LIN {X 0,Y 238.565,Z 456.874,A -85,B 0,C 180,E1 -19550.701,E2 -19550.701} C_VEL
LIN {X 0,Y 241.685,Z 448.178,A -85,B 0,C 180,E1 -19554.022,E2 -19554.022} C_VEL
LIN {X 0,Y 244.667,Z 440.384,A -85,B 0,C 180,E1 -19556.437,E2 -19556.437} C_VEL
LIN {X 0,Y 247.814,Z 431.182,A -85,B 0,C 180,E1 -19558.823,E2 -19558.823} C_VEL
LIN {X 0,Y 251.41,Z 420.34,A -85,B 0,C 180,E1 -19561.14,E2 -19561.14} C_VEL
LIN {X 0,Y 255.12,Z 408.504,A -85,B 0,C 180,E1 -19563.195,E2 -19563.195} C_VEL
LIN {X 0,Y 257.974,Z 398.718,A -85,B 0,C 180,E1 -19564.607,E2 -19564.607} C_VEL
LIN {X 0,Y 257.894,Z 393.482,A -85,B 0,C 180,E1 -19565.491,E2 -19565.491} C_VEL
LIN {X 0,Y 256.687,Z 381.828,A -85,B 0,C 180,E1 -19567.439,E2 -19567.439} C_VEL
LIN {X 0,Y 254.25,Z 368.563,A -85,B 0,C 180,E1 -19569.568,E2 -19569.568} C_VEL
LIN {X 0,Y 250.278,Z 354.47,A -85,B 0,C 180,E1 -19571.817,E2 -19571.817} C_VEL
LIN {X 0,Y 245.396,Z 341.798,A -85,B 0,C 180,E1 -19573.907,E2 -19573.907} C_VEL
LIN {X 0,Y 241.213,Z 333.323,A -85,B 0,C 180,E1 -19575.435,E2 -19575.435} C_VEL
LIN {X 0,Y 239.306,Z 329.7,A -85,B 0,C 180,E1 -19576.09,E2 -19576.09} C_VEL
LIN {X 0,Y 236.728,Z 325.904,A -85,B 0,C 180,E1 -19576.935,E2 -19576.935} C_VEL
LIN {X 0,Y 236.107,Z 323.82,A -85,B 0,C 180,E1 -19577.26,E2 -19577.26} C_VEL
LIN {X 0,Y 235.752,Z 321.234,A -85,B 0,C 180,E1 -19581.242,E2 -19581.242} C_VEL
LIN {X 0,Y 235.353,Z 318.757,A -85,B 0,C 180,E1 -19585.433,E2 -19585.433} C_VEL
LIN {X 0,Y 235.026,Z 316.609,A -85,B 0,C 180,E1 -19589.446,E2 -19589.446} C_VEL
LIN {X 0,Y 234.932,Z 315.851,A -85,B 0,C 180,E1 -19591.404,E2 -19591.404} C_VEL
LIN {X 0,Y 234.982,Z 315.842,A -85,B 0,C 180,E1 -19595.246,E2 -19595.246} C_VEL
LIN {X 0,Y 235.006,Z 315.837,A -85,B 0,C 180,E1 -19598.97,E2 -19598.97} C_VEL
LIN {X 0,Y 235.091,Z 315.823,A -85,B 0,C 180,E1 -19603.059,E2 -19603.059} C_VEL
LIN {X 0,Y 235.103,Z 315.821,A -85,B 0,C 180,E1 -19607.922,E2 -19607.922} C_VEL
LIN {X 0,Y 235.305,Z 315.795,A -85,B 0,C 180,E1 -19611.412,E2 -19611.412} C_VEL
LIN {X 0,Y 235.2,Z 315.808,A -85,B 0,C 180,E1 -19614.857,E2 -19614.857} C_VEL
LIN {X 0,Y 235.588,Z 315.759,A -85,B 0,C 180,E1 -19618.291,E2 -19618.291} C_VEL
LIN {X 0,Y 235.588,Z 315.764,A -85,B 0,C 180,E1 -19621.71,E2 -19621.71} C_VEL
LIN {X 0,Y 235.344,Z 315.795,A -85,B 0,C 180,E1 -19626.861,E2 -19626.861} C_VEL
LIN {X 0,Y 235.208,Z 315.813,A -85,B 0,C 180,E1 -19630.328,E2 -19630.328} C_VEL
LIN {X 0,Y 235.107,Z 315.822,A -85,B 0,C 180,E1 -19635.607,E2 -19635.607} C_VEL
LIN {X 0,Y 235.004,Z 315.838,A -85,B 0,C 180,E1 -19639.206,E2 -19639.206} C_VEL
LIN {X 0,Y 234.956,Z 315.845,A -85,B 0,C 180,E1 -19642.883,E2 -19642.883} C_VEL
LIN {X 0,Y 234.963,Z 315.84,A -85,B 0,C 180,E1 -19646.658,E2 -19646.658} C_VEL
LIN {X 0,Y 234.918,Z 315.843,A -85,B 0,C 180,E1 -19650.57,E2 -19650.57} C_VEL
LIN {X 0,Y 234.939,Z 315.84,A -85,B 0,C 180,E1 -19653.115,E2 -19653.115} C_VEL
LIN {X 0,Y 235.197,Z 317.589,A -85,B 0,C 180,E1 -19656.7,E2 -19656.7} C_VEL
LIN {X 0,Y 235.53,Z 319.939,A -85,B 0,C 180,E1 -19661.031,E2 -19661.031} C_VEL
LIN {X 0,Y 235.683,Z 321.16,A -85,B 0,C 180,E1 -19662.76,E2 -19662.76} C_VEL
LIN {X 0,Y 236.839,Z 324.025,A -85,B 0,C 180,E1 -19663.204,E2 -19663.204} C_VEL
LIN {X 0,Y 238.973,Z 326.929,A -85,B 0,C 180,E1 -19663.895,E2 -19663.895} C_VEL
LIN {X 0,Y 240.953,Z 330.465,A -85,B 0,C 180,E1 -19664.575,E2 -19664.575} C_VEL
LIN {X 0,Y 245.815,Z 339.929,A -85,B 0,C 180,E1 -19666.354,E2 -19666.354} C_VEL
LIN {X 0,Y 250.518,Z 351.507,A -85,B 0,C 180,E1 -19668.337,E2 -19668.337} C_VEL
LIN {X 0,Y 254.323,Z 363.793,A -85,B 0,C 180,E1 -19670.381,E2 -19670.381} C_VEL
LIN {X 0,Y 257.065,Z 376.3,A -85,B 0,C 180,E1 -19672.452,E2 -19672.452} C_VEL
LIN {X 0,Y 258.779,Z 388.609,A -85,B 0,C 180,E1 -19674.563,E2 -19674.563} C_VEL
LIN {X 0,Y 258.908,Z 392.584,A -85,B 0,C 180,E1 -19675.248,E2 -19675.248} C_VEL
LIN {X 0,Y 255.3,Z 405.294,A -85,B 0,C 180,E1 -19677.066,E2 -19677.066} C_VEL
LIN {X 0,Y 251.996,Z 415.961,A -85,B 0,C 180,E1 -19678.94,E2 -19678.94} C_VEL
LIN {X 0,Y 248.366,Z 427.006,A -85,B 0,C 180,E1 -19681.307,E2 -19681.307} C_VEL
LIN {X 0,Y 244.682,Z 437.336,A -85,B 0,C 180,E1 -19684.023,E2 -19684.023} C_VEL
LIN {X 0,Y 241.427,Z 446.098,A -85,B 0,C 180,E1 -19686.86,E2 -19686.86} C_VEL
LIN {X 0,Y 239.063,Z 452.429,A -85,B 0,C 180,E1 -19689.344,E2 -19689.344} C_VEL
LIN {X 0,Y 236.617,Z 459.393,A -85,B 0,C 180,E1 -19692.722,E2 -19692.722} C_VEL
LIN {X 0,Y 234.756,Z 464.865,A -85,B 0,C 180,E1 -19696.144,E2 -19696.144} C_VEL
LIN {X 0,Y 233.633,Z 468.994,A -85,B 0,C 180,E1 -19699.603,E2 -19699.603} C_VEL
LIN {X 0,Y 232.937,Z 471.894,A -85,B 0,C 180,E1 -19703.069,E2 -19703.069} C_VEL
LIN {X 0,Y 232.691,Z 473.635,A -85,B 0,C 180,E1 -19706.538,E2 -19706.538} C_VEL
LIN {X 0,Y 232.72,Z 474.241,A -85,B 0,C 180,E1 -19710.001,E2 -19710.001} C_VEL
LIN {X 0,Y 232.691,Z 473.672,A -85,B 0,C 180,E1 -19713.464,E2 -19713.464} C_VEL
LIN {X 0,Y 232.921,Z 471.98,A -85,B 0,C 180,E1 -19716.933,E2 -19716.933} C_VEL
LIN {X 0,Y 233.606,Z 469.125,A -85,B 0,C 180,E1 -19720.4,E2 -19720.4} C_VEL
LIN {X 0,Y 234.736,Z 465.04,A -85,B 0,C 180,E1 -19723.859,E2 -19723.859} C_VEL
LIN {X 0,Y 236.558,Z 459.624,A -85,B 0,C 180,E1 -19727.284,E2 -19727.284} C_VEL
LIN {X 0,Y 239.001,Z 452.724,A -85,B 0,C 180,E1 -19730.663,E2 -19730.663} C_VEL
LIN {X 0,Y 242.204,Z 444.112,A -85,B 0,C 180,E1 -19733.969,E2 -19733.969} C_VEL
LIN {X 0,Y 245.639,Z 434.956,A -85,B 0,C 180,E1 -19736.784,E2 -19736.784} C_VEL
LIN {X 0,Y 248.854,Z 425.634,A -85,B 0,C 180,E1 -19739.155,E2 -19739.155} C_VEL
LIN {X 0,Y 252.888,Z 413.567,A -85,B 0,C 180,E1 -19741.638,E2 -19741.638} C_VEL
LIN {X 0,Y 256.604,Z 401.244,A -85,B 0,C 180,E1 -19743.684,E2 -19743.684} C_VEL
LIN {X 0,Y 259.081,Z 391.806,A -85,B 0,C 180,E1 -19744.989,E2 -19744.989} C_VEL
LIN {X 0,Y 257.665,Z 379.68,A -85,B 0,C 180,E1 -19747.112,E2 -19747.112} C_VEL
LIN {X 0,Y 255.437,Z 368.067,A -85,B 0,C 180,E1 -19749.052,E2 -19749.052} C_VEL
LIN {X 0,Y 251.911,Z 355.507,A -85,B 0,C 180,E1 -19751.126,E2 -19751.126} C_VEL
LIN {X 0,Y 247.397,Z 343.495,A -85,B 0,C 180,E1 -19753.173,E2 -19753.173} C_VEL
LIN {X 0,Y 244.519,Z 337.246,A -85,B 0,C 180,E1 -19754.3,E2 -19754.3} C_VEL
LIN {X 0,Y 240.718,Z 330.109,A -85,B 0,C 180,E1 -19755.662,E2 -19755.662} C_VEL
LIN {X 0,Y 238.456,Z 326.031,A -85,B 0,C 180,E1 -19756.441,E2 -19756.441} C_VEL
LIN {X 0,Y 236.365,Z 323.227,A -85,B 0,C 180,E1 -19757.123,E2 -19757.123} C_VEL
LIN {X 0,Y 235.632,Z 320.937,A -85,B 0,C 180,E1 -19757.444,E2 -19757.444} C_VEL
LIN {X 0,Y 235.376,Z 318.821,A -85,B 0,C 180,E1 -19761.168,E2 -19761.168} C_VEL
LIN {X 0,Y 235.047,Z 316.644,A -85,B 0,C 180,E1 -19765.381,E2 -19765.381} C_VEL
LIN {X 0,Y 234.953,Z 315.845,A -85,B 0,C 180,E1 -19767.423,E2 -19767.423} C_VEL
LIN {X 0,Y 234.902,Z 315.849,A -85,B 0,C 180,E1 -19771.399,E2 -19771.399} C_VEL
LIN {X 0,Y 234.953,Z 315.841,A -85,B 0,C 180,E1 -19775.243,E2 -19775.243} C_VEL
LIN {X 0,Y 234.997,Z 315.838,A -85,B 0,C 180,E1 -19778.968,E2 -19778.968} C_VEL
LIN {X 0,Y 235.097,Z 315.822,A -85,B 0,C 180,E1 -19783.059,E2 -19783.059} C_VEL
LIN {X 0,Y 235.103,Z 315.821,A -85,B 0,C 180,E1 -19787.921,E2 -19787.921} C_VEL
LIN {X 0,Y 235.311,Z 315.798,A -85,B 0,C 180,E1 -19791.411,E2 -19791.411} C_VEL
LIN {X 0,Y 235.205,Z 315.813,A -85,B 0,C 180,E1 -19794.857,E2 -19794.857} C_VEL
LIN {X 0,Y 235.593,Z 315.765,A -85,B 0,C 180,E1 -19798.29,E2 -19798.29} C_VEL
LIN {X 0,Y 235.593,Z 315.764,A -85,B 0,C 180,E1 -19801.709,E2 -19801.709} C_VEL
LIN {X 0,Y 235.354,Z 315.792,A -85,B 0,C 180,E1 -19806.86,E2 -19806.86} C_VEL
LIN {X 0,Y 235.214,Z 315.812,A -85,B 0,C 180,E1 -19810.327,E2 -19810.327} C_VEL
LIN {X 0,Y 235.113,Z 315.824,A -85,B 0,C 180,E1 -19815.606,E2 -19815.606} C_VEL
LIN {X 0,Y 235.007,Z 315.837,A -85,B 0,C 180,E1 -19819.206,E2 -19819.206} C_VEL
LIN {X 0,Y 234.952,Z 315.844,A -85,B 0,C 180,E1 -19822.884,E2 -19822.884} C_VEL
LIN {X 0,Y 234.967,Z 315.843,A -85,B 0,C 180,E1 -19826.657,E2 -19826.657} C_VEL
LIN {X 0,Y 234.936,Z 315.851,A -85,B 0,C 180,E1 -19828.596,E2 -19828.596} C_VEL
LIN {X 0,Y 235.236,Z 317.68,A -85,B 0,C 180,E1 -19832.532,E2 -19832.532} C_VEL
LIN {X 0,Y 235.552,Z 319.993,A -85,B 0,C 180,E1 -19836.636,E2 -19836.636} C_VEL
LIN {X 0,Y 235.948,Z 322.582,A -85,B 0,C 180,E1 -19840.793,E2 -19840.793} C_VEL
LIN {X 0,Y 236.179,Z 323.866,A -85,B 0,C 180,E1 -19841.659,E2 -19841.659} C_VEL
LIN {X 0,Y 236.561,Z 326.147,A -85,B 0,C 180,E1 -19842.401,E2 -19842.401} C_VEL
LIN {X 0,Y 237.321,Z 330.696,A -85,B 0,C 180,E1 -19843.304,E2 -19843.304} C_VEL
LIN {X 0,Y 240.561,Z 345.361,A -85,B 0,C 180,E1 -19845.198,E2 -19845.198} C_VEL
LIN {X 0,Y 241.142,Z 347.057,A -85,B 0,C 180,E1 -19845.474,E2 -19845.474} C_VEL
LIN {X 0,Y 244.976,Z 357.702,A -85,B 0,C 180,E1 -19847.338,E2 -19847.338} C_VEL
LIN {X 0,Y 248.398,Z 370.303,A -85,B 0,C 180,E1 -19849.467,E2 -19849.467} C_VEL
LIN {X 0,Y 250.733,Z 383.447,A -85,B 0,C 180,E1 -19851.705,E2 -19851.705} C_VEL
LIN {X 0,Y 251.803,Z 394.831,A -85,B 0,C 180,E1 -19853.714,E2 -19853.714} C_VEL
LIN {X 0,Y 251.861,Z 399.873,A -85,B 0,C 180,E1 -19854.61,E2 -19854.61} C_VEL
LIN {X 0,Y 248.134,Z 412.127,A -85,B 0,C 180,E1 -19856.475,E2 -19856.475} C_VEL
LIN {X 0,Y 244.065,Z 424.3,A -85,B 0,C 180,E1 -19858.78,E2 -19858.78} C_VEL
LIN {X 0,Y 240.312,Z 434.52,A -85,B 0,C 180,E1 -19861.149,E2 -19861.149} C_VEL
LIN {X 0,Y 236.728,Z 444.502,A -85,B 0,C 180,E1 -19864.03,E2 -19864.03} C_VEL
LIN {X 0,Y 233.466,Z 452.792,A -85,B 0,C 180,E1 -19866.962,E2 -19866.962} C_VEL
LIN {X 0,Y 230.488,Z 460.579,A -85,B 0,C 180,E1 -19870.402,E2 -19870.402} C_VEL
LIN {X 0,Y 228.359,Z 466.775,A -85,B 0,C 180,E1 -19873.919,E2 -19873.919} C_VEL
LIN {X 0,Y 226.816,Z 471.566,A -85,B 0,C 180,E1 -19877.473,E2 -19877.473} C_VEL
LIN {X 0,Y 225.98,Z 475.077,A -85,B 0,C 180,E1 -19881.054,E2 -19881.054} C_VEL
LIN {X 0,Y 225.589,Z 477.385,A -85,B 0,C 180,E1 -19884.637,E2 -19884.637} C_VEL
LIN {X 0,Y 225.545,Z 478.545,A -85,B 0,C 180,E1 -19888.214,E2 -19888.214} C_VEL
LIN {X 0,Y 225.631,Z 478.698,A -85,B 0,C 180,E1 -19889.999,E2 -19889.999} C_VEL
LIN {X 0,Y 225.522,Z 478.094,A -85,B 0,C 180,E1 -19893.573,E2 -19893.573} C_VEL
LIN {X 0,Y 225.734,Z 476.348,A -85,B 0,C 180,E1 -19897.153,E2 -19897.153} C_VEL
LIN {X 0,Y 226.336,Z 473.435,A -85,B 0,C 180,E1 -19900.736,E2 -19900.736} C_VEL
LIN {X 0,Y 227.557,Z 469.287,A -85,B 0,C 180,E1 -19904.304,E2 -19904.304} C_VEL
LIN {X 0,Y 229.363,Z 463.793,A -85,B 0,C 180,E1 -19907.842,E2 -19907.842} C_VEL
LIN {X 0,Y 231.889,Z 456.803,A -85,B 0,C 180,E1 -19911.326,E2 -19911.326} C_VEL
LIN {X 0,Y 235.171,Z 448.107,A -85,B 0,C 180,E1 -19914.732,E2 -19914.732} C_VEL
LIN {X 0,Y 238.269,Z 440.313,A -85,B 0,C 180,E1 -19917.205,E2 -19917.205} C_VEL
LIN {X 0,Y 242.163,Z 429.475,A -85,B 0,C 180,E1 -19920.04,E2 -19920.04} C_VEL
LIN {X 0,Y 246.341,Z 417.287,A -85,B 0,C 180,E1 -19922.58,E2 -19922.58} C_VEL
LIN {X 0,Y 250.239,Z 405.245,A -85,B 0,C 180,E1 -19924.586,E2 -19924.586} C_VEL
LIN {X 0,Y 251.755,Z 399.909,A -85,B 0,C 180,E1 -19925.354,E2 -19925.354} C_VEL
LIN {X 0,Y 251.35,Z 389.821,A -85,B 0,C 180,E1 -19927.147,E2 -19927.147} C_VEL
LIN {X 0,Y 249.87,Z 378.381,A -85,B 0,C 180,E1 -19929.135,E2 -19929.135} C_VEL
LIN {X 0,Y 247.702,Z 367.848,A -85,B 0,C 180,E1 -19930.905,E2 -19930.905} C_VEL
LIN {X 0,Y 244.696,Z 356.943,A -85,B 0,C 180,E1 -19932.745,E2 -19932.745} C_VEL
LIN {X 0,Y 240.512,Z 345.764,A -85,B 0,C 180,E1 -19934.713,E2 -19934.713} C_VEL
LIN {X 0,Y 236.668,Z 337.699,A -85,B 0,C 180,E1 -19936.263,E2 -19936.263} C_VEL
LIN {X 0,Y 234.508,Z 333.706,A -85,B 0,C 180,E1 -19937.089,E2 -19937.089} C_VEL
LIN {X 0,Y 232.407,Z 330.075,A -85,B 0,C 180,E1 -19937.86,E2 -19937.86} C_VEL
LIN {X 0,Y 231.653,Z 328.876,A -85,B 0,C 180,E1 -19938.13,E2 -19938.13} C_VEL
LIN {X 0,Y 229.64,Z 325.946,A -85,B 0,C 180,E1 -19938.853,E2 -19938.853} C_VEL
LIN {X 0,Y 228.973,Z 323.734,A -85,B 0,C 180,E1 -19939.217,E2 -19939.217} C_VEL
LIN {X 0,Y 228.476,Z 320.749,A -85,B 0,C 180,E1 -19944.236,E2 -19944.236} C_VEL
LIN {X 0,Y 228.14,Z 318.506,A -85,B 0,C 180,E1 -19948.42,E2 -19948.42} C_VEL
LIN {X 0,Y 227.874,Z 316.729,A -85,B 0,C 180,E1 -19952.444,E2 -19952.444} C_VEL
LIN {X 0,Y 227.909,Z 316.72,A -85,B 0,C 180,E1 -19956.367,E2 -19956.367} C_VEL
LIN {X 0,Y 227.937,Z 316.715,A -85,B 0,C 180,E1 -19960.174,E2 -19960.174} C_VEL
LIN {X 0,Y 228.051,Z 316.704,A -85,B 0,C 180,E1 -19963.898,E2 -19963.898} C_VEL
LIN {X 0,Y 228.062,Z 316.699,A -85,B 0,C 180,E1 -19967.543,E2 -19967.543} C_VEL
LIN {X 0,Y 228.246,Z 316.674,A -85,B 0,C 180,E1 -19971.144,E2 -19971.144} C_VEL
LIN {X 0,Y 228.296,Z 316.673,A -85,B 0,C 180,E1 -19972.927,E2 -19972.927} C_VEL
LIN {X 0,Y 228.547,Z 316.636,A -85,B 0,C 180,E1 -19978.238,E2 -19978.238} C_VEL
LIN {X 0,Y 228.547,Z 316.641,A -85,B 0,C 180,E1 -19981.762,E2 -19981.762} C_VEL
LIN {X 0,Y 228.296,Z 316.673,A -85,B 0,C 180,E1 -19987.073,E2 -19987.073} C_VEL
LIN {X 0,Y 228.139,Z 316.69,A -85,B 0,C 180,E1 -19990.652,E2 -19990.652} C_VEL
LIN {X 0,Y 228.055,Z 316.699,A -85,B 0,C 180,E1 -19994.273,E2 -19994.273} C_VEL
LIN {X 0,Y 227.998,Z 316.706,A -85,B 0,C 180,E1 -19997.954,E2 -19997.954} C_VEL
LIN {X 0,Y 227.925,Z 316.719,A -85,B 0,C 180,E1 -20002.33,E2 -20002.33} C_VEL
LIN {X 0,Y 227.937,Z 316.715,A -85,B 0,C 180,E1 -20006.603,E2 -20006.603} C_VEL
LIN {X 0,Y 227.893,Z 316.717,A -85,B 0,C 180,E1 -20010.292,E2 -20010.292} C_VEL
LIN {X 0,Y 227.862,Z 316.722,A -85,B 0,C 180,E1 -20011.624,E2 -20011.624} C_VEL
LIN {X 0,Y 228.139,Z 318.464,A -85,B 0,C 180,E1 -20015.825,E2 -20015.825} C_VEL
LIN {X 0,Y 228.495,Z 320.901,A -85,B 0,C 180,E1 -20020.524,E2 -20020.524} C_VEL
LIN {X 0,Y 228.578,Z 321.271,A -85,B 0,C 180,E1 -20020.796,E2 -20020.796} C_VEL
LIN {X 0,Y 229.838,Z 324.342,A -85,B 0,C 180,E1 -20021.323,E2 -20021.323} C_VEL
LIN {X 0,Y 231.924,Z 327.058,A -85,B 0,C 180,E1 -20022.054,E2 -20022.054} C_VEL
LIN {X 0,Y 234.094,Z 330.783,A -85,B 0,C 180,E1 -20022.859,E2 -20022.859} C_VEL
LIN {X 0,Y 235.185,Z 332.597,A -85,B 0,C 180,E1 -20023.27,E2 -20023.27} C_VEL
LIN {X 0,Y 239.558,Z 340.943,A -85,B 0,C 180,E1 -20024.983,E2 -20024.983} C_VEL
LIN {X 0,Y 243.811,Z 350.913,A -85,B 0,C 180,E1 -20026.854,E2 -20026.854} C_VEL
LIN {X 0,Y 247.435,Z 362.038,A -85,B 0,C 180,E1 -20028.826,E2 -20028.826} C_VEL
LIN {X 0,Y 250.277,Z 373.956,A -85,B 0,C 180,E1 -20030.896,E2 -20030.896} C_VEL
LIN {X 0,Y 252.067,Z 385.053,A -85,B 0,C 180,E1 -20032.884,E2 -20032.884} C_VEL
LIN {X 0,Y 252.732,Z 394.02,A -85,B 0,C 180,E1 -20034.505,E2 -20034.505} C_VEL
LIN {X 0,Y 248.996,Z 406.539,A -85,B 0,C 180,E1 -20036.365,E2 -20036.365} C_VEL
LIN {X 0,Y 245.266,Z 417.98,A -85,B 0,C 180,E1 -20038.471,E2 -20038.471} C_VEL
LIN {X 0,Y 241.896,Z 427.696,A -85,B 0,C 180,E1 -20040.647,E2 -20040.647} C_VEL
LIN {X 0,Y 238.299,Z 437.407,A -85,B 0,C 180,E1 -20043.273,E2 -20043.273} C_VEL
LIN {X 0,Y 234.867,Z 446.17,A -85,B 0,C 180,E1 -20046.175,E2 -20046.175} C_VEL
LIN {X 0,Y 232.386,Z 452.5,A -85,B 0,C 180,E1 -20048.722,E2 -20048.722} C_VEL
LIN {X 0,Y 229.807,Z 459.464,A -85,B 0,C 180,E1 -20052.193,E2 -20052.193} C_VEL
LIN {X 0,Y 227.837,Z 464.935,A -85,B 0,C 180,E1 -20055.714,E2 -20055.714} C_VEL
LIN {X 0,Y 226.612,Z 469.064,A -85,B 0,C 180,E1 -20059.277,E2 -20059.277} C_VEL
LIN {X 0,Y 225.885,Z 471.963,A -85,B 0,C 180,E1 -20062.852,E2 -20062.852} C_VEL
LIN {X 0,Y 225.606,Z 473.704,A -85,B 0,C 180,E1 -20066.429,E2 -20066.429} C_VEL
LIN {X 0,Y 225.636,Z 474.31,A -85,B 0,C 180,E1 -20070.001,E2 -20070.001} C_VEL
LIN {X 0,Y 225.605,Z 473.741,A -85,B 0,C 180,E1 -20073.573,E2 -20073.573} C_VEL
LIN {X 0,Y 225.845,Z 472.049,A -85,B 0,C 180,E1 -20077.151,E2 -20077.151} C_VEL
LIN {X 0,Y 226.586,Z 469.194,A -85,B 0,C 180,E1 -20080.726,E2 -20080.726} C_VEL
LIN {X 0,Y 227.816,Z 465.108,A -85,B 0,C 180,E1 -20084.288,E2 -20084.288} C_VEL
LIN {X 0,Y 229.751,Z 459.692,A -85,B 0,C 180,E1 -20087.812,E2 -20087.812} C_VEL
LIN {X 0,Y 232.335,Z 452.792,A -85,B 0,C 180,E1 -20091.284,E2 -20091.284} C_VEL
LIN {X 0,Y 235.672,Z 444.18,A -85,B 0,C 180,E1 -20094.677,E2 -20094.677} C_VEL
LIN {X 0,Y 239.29,Z 435.023,A -85,B 0,C 180,E1 -20097.554,E2 -20097.554} C_VEL
LIN {X 0,Y 242.649,Z 425.701,A -85,B 0,C 180,E1 -20099.975,E2 -20099.975} C_VEL
LIN {X 0,Y 246.85,Z 413.633,A -85,B 0,C 180,E1 -20102.506,E2 -20102.506} C_VEL
LIN {X 0,Y 250.725,Z 401.309,A -85,B 0,C 180,E1 -20104.585,E2 -20104.585} C_VEL
LIN {X 0,Y 252.885,Z 393.447,A -85,B 0,C 180,E1 -20105.705,E2 -20105.705} C_VEL
LIN {X 0,Y 251.603,Z 381.432,A -85,B 0,C 180,E1 -20107.917,E2 -20107.917} C_VEL
LIN {X 0,Y 249.779,Z 371.284,A -85,B 0,C 180,E1 -20109.695,E2 -20109.695} C_VEL
LIN {X 0,Y 246.555,Z 358.913,A -85,B 0,C 180,E1 -20111.867,E2 -20111.867} C_VEL
LIN {X 0,Y 242.119,Z 346.554,A -85,B 0,C 180,E1 -20114.09,E2 -20114.09} C_VEL
LIN {X 0,Y 238.454,Z 338.74,A -85,B 0,C 180,E1 -20115.623,E2 -20115.623} C_VEL
LIN {X 0,Y 236.232,Z 334.554,A -85,B 0,C 180,E1 -20116.487,E2 -20116.487} C_VEL
LIN {X 0,Y 234.378,Z 331.128,A -85,B 0,C 180,E1 -20117.206,E2 -20117.206} C_VEL
LIN {X 0,Y 232.191,Z 327.696,A -85,B 0,C 180,E1 -20118.005,E2 -20118.005} C_VEL
LIN {X 0,Y 231.476,Z 326.274,A -85,B 0,C 180,E1 -20118.28,E2 -20118.28} C_VEL
LIN {X 0,Y 229.392,Z 323.598,A -85,B 0,C 180,E1 -20119.017,E2 -20119.017} C_VEL
LIN {X 0,Y 228.507,Z 321.026,A -85,B 0,C 180,E1 -20119.443,E2 -20119.443} C_VEL
LIN {X 0,Y 228.159,Z 318.562,A -85,B 0,C 180,E1 -20124.179,E2 -20124.179} C_VEL
LIN {X 0,Y 227.856,Z 316.73,A -85,B 0,C 180,E1 -20128.375,E2 -20128.375} C_VEL
LIN {X 0,Y 227.855,Z 316.728,A -85,B 0,C 180,E1 -20132.441,E2 -20132.441} C_VEL
LIN {X 0,Y 227.895,Z 316.723,A -85,B 0,C 180,E1 -20136.365,E2 -20136.365} C_VEL
LIN {X 0,Y 227.937,Z 316.714,A -85,B 0,C 180,E1 -20140.174,E2 -20140.174} C_VEL
LIN {X 0,Y 228.058,Z 316.697,A -85,B 0,C 180,E1 -20143.898,E2 -20143.898} C_VEL
LIN {X 0,Y 228.063,Z 316.695,A -85,B 0,C 180,E1 -20147.542,E2 -20147.542} C_VEL
LIN {X 0,Y 228.252,Z 316.678,A -85,B 0,C 180,E1 -20151.144,E2 -20151.144} C_VEL
LIN {X 0,Y 228.302,Z 316.672,A -85,B 0,C 180,E1 -20152.927,E2 -20152.927} C_VEL
LIN {X 0,Y 228.552,Z 316.641,A -85,B 0,C 180,E1 -20158.238,E2 -20158.238} C_VEL
LIN {X 0,Y 228.552,Z 316.641,A -85,B 0,C 180,E1 -20161.762,E2 -20161.762} C_VEL
LIN {X 0,Y 228.307,Z 316.67,A -85,B 0,C 180,E1 -20167.073,E2 -20167.073} C_VEL
LIN {X 0,Y 228.145,Z 316.692,A -85,B 0,C 180,E1 -20170.651,E2 -20170.651} C_VEL
LIN {X 0,Y 228.064,Z 316.702,A -85,B 0,C 180,E1 -20174.272,E2 -20174.272} C_VEL
LIN {X 0,Y 228.002,Z 316.71,A -85,B 0,C 180,E1 -20177.953,E2 -20177.953} C_VEL
LIN {X 0,Y 227.916,Z 316.72,A -85,B 0,C 180,E1 -20182.321,E2 -20182.321} C_VEL
LIN {X 0,Y 227.941,Z 316.718,A -85,B 0,C 180,E1 -20186.602,E2 -20186.602} C_VEL
LIN {X 0,Y 227.878,Z 316.728,A -85,B 0,C 180,E1 -20187.556,E2 -20187.556} C_VEL
LIN {X 0,Y 228.153,Z 318.556,A -85,B 0,C 180,E1 -20191.578,E2 -20191.578} C_VEL
LIN {X 0,Y 228.484,Z 320.799,A -85,B 0,C 180,E1 -20195.762,E2 -20195.762} C_VEL
LIN {X 0,Y 228.993,Z 323.937,A -85,B 0,C 180,E1 -20200.779,E2 -20200.779} C_VEL
LIN {X 0,Y 230.128,Z 326.9,A -85,B 0,C 180,E1 -20201.259,E2 -20201.259} C_VEL
LIN {X 0,Y 232.296,Z 329.791,A -85,B 0,C 180,E1 -20202.019,E2 -20202.019} C_VEL
LIN {X 0,Y 234.381,Z 333.546,A -85,B 0,C 180,E1 -20202.793,E2 -20202.793} C_VEL
LIN {X 0,Y 235.827,Z 336.082,A -85,B 0,C 180,E1 -20203.343,E2 -20203.343} C_VEL
LIN {X 0,Y 239.693,Z 343.792,A -85,B 0,C 180,E1 -20204.869,E2 -20204.869} C_VEL
LIN {X 0,Y 241.142,Z 347.057,A -85,B 0,C 180,E1 -20205.474,E2 -20205.474} C_VEL
LIN {X 0,Y 242.393,Z 351.967,A -85,B 0,C 180,E1 -20206.193,E2 -20206.193} C_VEL
LIN {X 0,Y 242.772,Z 360.897,A -85,B 0,C 180,E1 -20207.207,E2 -20207.207} C_VEL
LIN {X 0,Y 242.613,Z 368.127,A -85,B 0,C 180,E1 -20208.029,E2 -20208.029} C_VEL
LIN {X 0,Y 243.089,Z 374.88,A -85,B 0,C 180,E1 -20209.021,E2 -20209.021} C_VEL
LIN {X 0,Y 244.917,Z 386.896,A -85,B 0,C 180,E1 -20211.179,E2 -20211.179} C_VEL
LIN {X 0,Y 245.705,Z 397.844,A -85,B 0,C 180,E1 -20213.215,E2 -20213.215} C_VEL
LIN {X 0,Y 245.682,Z 401.141,A -85,B 0,C 180,E1 -20213.842,E2 -20213.842} C_VEL
LIN {X 0,Y 241.853,Z 413.132,A -85,B 0,C 180,E1 -20215.735,E2 -20215.735} C_VEL
LIN {X 0,Y 237.987,Z 424.233,A -85,B 0,C 180,E1 -20217.889,E2 -20217.889} C_VEL
LIN {X 0,Y 234.084,Z 434.453,A -85,B 0,C 180,E1 -20220.306,E2 -20220.306} C_VEL
LIN {X 0,Y 230.314,Z 444.434,A -85,B 0,C 180,E1 -20223.25,E2 -20223.25} C_VEL
LIN {X 0,Y 226.909,Z 452.724,A -85,B 0,C 180,E1 -20226.256,E2 -20226.256} C_VEL
LIN {X 0,Y 223.745,Z 460.511,A -85,B 0,C 180,E1 -20229.786,E2 -20229.786} C_VEL
LIN {X 0,Y 221.477,Z 466.706,A -85,B 0,C 180,E1 -20233.405,E2 -20233.405} C_VEL
LIN {X 0,Y 219.84,Z 471.497,A -85,B 0,C 180,E1 -20237.068,E2 -20237.068} C_VEL
LIN {X 0,Y 218.942,Z 475.008,A -85,B 0,C 180,E1 -20240.764,E2 -20240.764} C_VEL
LIN {X 0,Y 218.5,Z 477.316,A -85,B 0,C 180,E1 -20244.462,E2 -20244.462} C_VEL
LIN {X 0,Y 218.448,Z 478.476,A -85,B 0,C 180,E1 -20248.156,E2 -20248.156} C_VEL
LIN {X 0,Y 218.53,Z 478.629,A -85,B 0,C 180,E1 -20249.999,E2 -20249.999} C_VEL
LIN {X 0,Y 218.427,Z 477.911,A -85,B 0,C 180,E1 -20254.104,E2 -20254.104} C_VEL
LIN {X 0,Y 218.653,Z 476.278,A -85,B 0,C 180,E1 -20257.386,E2 -20257.386} C_VEL
LIN {X 0,Y 219.307,Z 473.365,A -85,B 0,C 180,E1 -20261.085,E2 -20261.085} C_VEL
LIN {X 0,Y 220.619,Z 469.217,A -85,B 0,C 180,E1 -20264.764,E2 -20264.764} C_VEL
LIN {X 0,Y 222.54,Z 463.722,A -85,B 0,C 180,E1 -20268.409,E2 -20268.409} C_VEL
LIN {X 0,Y 225.223,Z 456.732,A -85,B 0,C 180,E1 -20271.99,E2 -20271.99} C_VEL
LIN {X 0,Y 228.713,Z 448.035,A -85,B 0,C 180,E1 -20275.479,E2 -20275.479} C_VEL
LIN {X 0,Y 231.906,Z 440.241,A -85,B 0,C 180,E1 -20278.016,E2 -20278.016} C_VEL
LIN {X 0,Y 235.992,Z 429.403,A -85,B 0,C 180,E1 -20280.91,E2 -20280.91} C_VEL
LIN {X 0,Y 240.359,Z 417.214,A -85,B 0,C 180,E1 -20283.496,E2 -20283.496} C_VEL
LIN {X 0,Y 244.31,Z 405.468,A -85,B 0,C 180,E1 -20285.489,E2 -20285.489} C_VEL
LIN {X 0,Y 245.578,Z 401.09,A -85,B 0,C 180,E1 -20286.137,E2 -20286.137} C_VEL
LIN {X 0,Y 245.139,Z 390.146,A -85,B 0,C 180,E1 -20288.188,E2 -20288.188} C_VEL
LIN {X 0,Y 243.619,Z 378.181,A -85,B 0,C 180,E1 -20290.359,E2 -20290.359} C_VEL
LIN {X 0,Y 241.034,Z 366.197,A -85,B 0,C 180,E1 -20292.487,E2 -20292.487} C_VEL
LIN {X 0,Y 237.382,Z 354.165,A -85,B 0,C 180,E1 -20294.676,E2 -20294.676} C_VEL
LIN {X 0,Y 233.977,Z 345.863,A -85,B 0,C 180,E1 -20296.303,E2 -20296.303} C_VEL
LIN {X 0,Y 230.381,Z 338.676,A -85,B 0,C 180,E1 -20297.846,E2 -20297.846} C_VEL
LIN {X 0,Y 227.567,Z 333.769,A -85,B 0,C 180,E1 -20298.991,E2 -20298.991} C_VEL
LIN {X 0,Y 225.577,Z 330.453,A -85,B 0,C 180,E1 -20299.785,E2 -20299.785} C_VEL
LIN {X 0,Y 224.793,Z 329.066,A -85,B 0,C 180,E1 -20300.101,E2 -20300.101} C_VEL
LIN {X 0,Y 222.568,Z 326.154,A -85,B 0,C 180,E1 -20300.962,E2 -20300.962} C_VEL
LIN {X 0,Y 221.711,Z 323.651,A -85,B 0,C 180,E1 -20301.407,E2 -20301.407} C_VEL
LIN {X 0,Y 221.383,Z 321.298,A -85,B 0,C 180,E1 -20305.626,E2 -20305.626} C_VEL
LIN {X 0,Y 221.105,Z 319.389,A -85,B 0,C 180,E1 -20309.431,E2 -20309.431} C_VEL
LIN {X 0,Y 220.889,Z 317.6,A -85,B 0,C 180,E1 -20313.549,E2 -20313.549} C_VEL
LIN {X 0,Y 220.873,Z 317.598,A -85,B 0,C 180,E1 -20317.553,E2 -20317.553} C_VEL
LIN {X 0,Y 220.979,Z 317.581,A -85,B 0,C 180,E1 -20322.571,E2 -20322.571} C_VEL
LIN {X 0,Y 221.002,Z 317.58,A -85,B 0,C 180,E1 -20327.138,E2 -20327.138} C_VEL
LIN {X 0,Y 221.188,Z 317.553,A -85,B 0,C 180,E1 -20330.859,E2 -20330.859} C_VEL
LIN {X 0,Y 221.121,Z 317.561,A -85,B 0,C 180,E1 -20334.529,E2 -20334.529} C_VEL
LIN {X 0,Y 221.505,Z 317.512,A -85,B 0,C 180,E1 -20338.182,E2 -20338.182} C_VEL
LIN {X 0,Y 221.505,Z 317.518,A -85,B 0,C 180,E1 -20341.818,E2 -20341.818} C_VEL
LIN {X 0,Y 221.234,Z 317.55,A -85,B 0,C 180,E1 -20347.3,E2 -20347.3} C_VEL
LIN {X 0,Y 221.06,Z 317.57,A -85,B 0,C 180,E1 -20350.997,E2 -20350.997} C_VEL
LIN {X 0,Y 221.011,Z 317.58,A -85,B 0,C 180,E1 -20356.63,E2 -20356.63} C_VEL
LIN {X 0,Y 220.888,Z 317.592,A -85,B 0,C 180,E1 -20360.487,E2 -20360.487} C_VEL
LIN {X 0,Y 220.863,Z 317.598,A -85,B 0,C 180,E1 -20364.436,E2 -20364.436} C_VEL
LIN {X 0,Y 220.823,Z 317.6,A -85,B 0,C 180,E1 -20368.516,E2 -20368.516} C_VEL
LIN {X 0,Y 220.835,Z 317.597,A -85,B 0,C 180,E1 -20370.768,E2 -20370.768} C_VEL
LIN {X 0,Y 221.073,Z 319.369,A -85,B 0,C 180,E1 -20374.906,E2 -20374.906} C_VEL
LIN {X 0,Y 221.382,Z 321.332,A -85,B 0,C 180,E1 -20378.584,E2 -20378.584} C_VEL
LIN {X 0,Y 222.505,Z 324.182,A -85,B 0,C 180,E1 -20379.108,E2 -20379.108} C_VEL
LIN {X 0,Y 225.015,Z 327.285,A -85,B 0,C 180,E1 -20380.071,E2 -20380.071} C_VEL
LIN {X 0,Y 226.995,Z 330.785,A -85,B 0,C 180,E1 -20380.882,E2 -20380.882} C_VEL
LIN {X 0,Y 228.278,Z 332.78,A -85,B 0,C 180,E1 -20381.4,E2 -20381.4} C_VEL
LIN {X 0,Y 231.304,Z 338.068,A -85,B 0,C 180,E1 -20382.635,E2 -20382.635} C_VEL
LIN {X 0,Y 235.398,Z 346.387,A -85,B 0,C 180,E1 -20384.437,E2 -20384.437} C_VEL
LIN {X 0,Y 239.556,Z 357.244,A -85,B 0,C 180,E1 -20386.572,E2 -20386.572} C_VEL
LIN {X 0,Y 242.91,Z 369.13,A -85,B 0,C 180,E1 -20388.785,E2 -20388.785} C_VEL
LIN {X 0,Y 245.334,Z 381.553,A -85,B 0,C 180,E1 -20391.087,E2 -20391.087} C_VEL
LIN {X 0,Y 246.592,Z 394.098,A -85,B 0,C 180,E1 -20393.481,E2 -20393.481} C_VEL
LIN {X 0,Y 246.588,Z 395.377,A -85,B 0,C 180,E1 -20393.717,E2 -20393.717} C_VEL
LIN {X 0,Y 242.751,Z 407.773,A -85,B 0,C 180,E1 -20395.63,E2 -20395.63} C_VEL
LIN {X 0,Y 238.545,Z 419.976,A -85,B 0,C 180,E1 -20397.975,E2 -20397.975} C_VEL
LIN {X 0,Y 234.831,Z 430.014,A -85,B 0,C 180,E1 -20400.357,E2 -20400.357} C_VEL
LIN {X 0,Y 230.801,Z 440.179,A -85,B 0,C 180,E1 -20403.312,E2 -20403.312} C_VEL
LIN {X 0,Y 227.429,Z 448.466,A -85,B 0,C 180,E1 -20406.315,E2 -20406.315} C_VEL
LIN {X 0,Y 224.304,Z 456.251,A -85,B 0,C 180,E1 -20409.84,E2 -20409.84} C_VEL
LIN {X 0,Y 221.948,Z 462.446,A -85,B 0,C 180,E1 -20413.443,E2 -20413.443} C_VEL
LIN {X 0,Y 220.176,Z 467.23,A -85,B 0,C 180,E1 -20417.09,E2 -20417.09} C_VEL
LIN {X 0,Y 219.129,Z 470.732,A -85,B 0,C 180,E1 -20420.773,E2 -20420.773} C_VEL
LIN {X 0,Y 218.601,Z 473.045,A -85,B 0,C 180,E1 -20424.466,E2 -20424.466} C_VEL
LIN {X 0,Y 218.489,Z 474.222,A -85,B 0,C 180,E1 -20428.157,E2 -20428.157} C_VEL
LIN {X 0,Y 218.536,Z 474.379,A -85,B 0,C 180,E1 -20430.001,E2 -20430.001} C_VEL
LIN {X 0,Y 218.504,Z 473.81,A -85,B 0,C 180,E1 -20433.689,E2 -20433.689} C_VEL
LIN {X 0,Y 218.795,Z 472.118,A -85,B 0,C 180,E1 -20437.383,E2 -20437.383} C_VEL
LIN {X 0,Y 219.584,Z 469.262,A -85,B 0,C 180,E1 -20441.072,E2 -20441.072} C_VEL
LIN {X 0,Y 220.916,Z 465.176,A -85,B 0,C 180,E1 -20444.745,E2 -20444.745} C_VEL
LIN {X 0,Y 222.954,Z 459.76,A -85,B 0,C 180,E1 -20448.375,E2 -20448.375} C_VEL
LIN {X 0,Y 225.687,Z 452.859,A -85,B 0,C 180,E1 -20451.943,E2 -20451.943} C_VEL
LIN {X 0,Y 229.186,Z 444.247,A -85,B 0,C 180,E1 -20455.424,E2 -20455.424} C_VEL
LIN {X 0,Y 232.984,Z 435.09,A -85,B 0,C 180,E1 -20458.366,E2 -20458.366} C_VEL
LIN {X 0,Y 236.491,Z 425.767,A -85,B 0,C 180,E1 -20460.84,E2 -20460.84} C_VEL
LIN {X 0,Y 240.849,Z 413.699,A -85,B 0,C 180,E1 -20463.42,E2 -20463.42} C_VEL
LIN {X 0,Y 244.839,Z 401.593,A -85,B 0,C 180,E1 -20465.495,E2 -20465.495} C_VEL
LIN {X 0,Y 246.608,Z 395.768,A -85,B 0,C 180,E1 -20466.342,E2 -20466.342} C_VEL
LIN {X 0,Y 245.919,Z 386.077,A -85,B 0,C 180,E1 -20468.196,E2 -20468.196} C_VEL
LIN {X 0,Y 244.255,Z 375.04,A -85,B 0,C 180,E1 -20470.263,E2 -20470.263} C_VEL
LIN {X 0,Y 241.179,Z 362.238,A -85,B 0,C 180,E1 -20472.625,E2 -20472.625} C_VEL
LIN {X 0,Y 236.697,Z 349.286,A -85,B 0,C 180,E1 -20475.111,E2 -20475.111} C_VEL
LIN {X 0,Y 232.649,Z 340.483,A -85,B 0,C 180,E1 -20476.958,E2 -20476.958} C_VEL
LIN {X 0,Y 229.811,Z 335.48,A -85,B 0,C 180,E1 -20478.139,E2 -20478.139} C_VEL
LIN {X 0,Y 227.348,Z 331.208,A -85,B 0,C 180,E1 -20479.156,E2 -20479.156} C_VEL
LIN {X 0,Y 225.189,Z 327.723,A -85,B 0,C 180,E1 -20480.027,E2 -20480.027} C_VEL
LIN {X 0,Y 224.496,Z 326.515,A -85,B 0,C 180,E1 -20480.309,E2 -20480.309} C_VEL
LIN {X 0,Y 222.352,Z 323.96,A -85,B 0,C 180,E1 -20481.134,E2 -20481.134} C_VEL
LIN {X 0,Y 221.358,Z 321.109,A -85,B 0,C 180,E1 -20481.682,E2 -20481.682} C_VEL
LIN {X 0,Y 221.073,Z 319.163,A -85,B 0,C 180,E1 -20485.746,E2 -20485.746} C_VEL
LIN {X 0,Y 220.835,Z 317.602,A -85,B 0,C 180,E1 -20489.389,E2 -20489.389} C_VEL
LIN {X 0,Y 220.876,Z 317.595,A -85,B 0,C 180,E1 -20493.547,E2 -20493.547} C_VEL
LIN {X 0,Y 220.868,Z 317.594,A -85,B 0,C 180,E1 -20497.552,E2 -20497.552} C_VEL
LIN {X 0,Y 220.985,Z 317.584,A -85,B 0,C 180,E1 -20502.571,E2 -20502.571} C_VEL
LIN {X 0,Y 221.003,Z 317.574,A -85,B 0,C 180,E1 -20507.138,E2 -20507.138} C_VEL
LIN {X 0,Y 221.194,Z 317.559,A -85,B 0,C 180,E1 -20510.859,E2 -20510.859} C_VEL
LIN {X 0,Y 221.125,Z 317.567,A -85,B 0,C 180,E1 -20514.528,E2 -20514.528} C_VEL
LIN {X 0,Y 221.51,Z 317.518,A -85,B 0,C 180,E1 -20518.182,E2 -20518.182} C_VEL
LIN {X 0,Y 221.509,Z 317.518,A -85,B 0,C 180,E1 -20521.818,E2 -20521.818} C_VEL
LIN {X 0,Y 221.244,Z 317.55,A -85,B 0,C 180,E1 -20527.3,E2 -20527.3} C_VEL
LIN {X 0,Y 221.067,Z 317.574,A -85,B 0,C 180,E1 -20530.996,E2 -20530.996} C_VEL
LIN {X 0,Y 220.995,Z 317.583,A -85,B 0,C 180,E1 -20534.739,E2 -20534.739} C_VEL
LIN {X 0,Y 220.92,Z 317.593,A -85,B 0,C 180,E1 -20538.549,E2 -20538.549} C_VEL
LIN {X 0,Y 220.884,Z 317.596,A -85,B 0,C 180,E1 -20542.675,E2 -20542.675} C_VEL
LIN {X 0,Y 220.893,Z 317.596,A -85,B 0,C 180,E1 -20546.45,E2 -20546.45} C_VEL
LIN {X 0,Y 221.141,Z 319.599,A -85,B 0,C 180,E1 -20550.899,E2 -20550.899} C_VEL
LIN {X 0,Y 221.419,Z 321.602,A -85,B 0,C 180,E1 -20554.843,E2 -20554.843} C_VEL
LIN {X 0,Y 221.706,Z 323.667,A -85,B 0,C 180,E1 -20558.532,E2 -20558.532} C_VEL
LIN {X 0,Y 222.903,Z 326.801,A -85,B 0,C 180,E1 -20559.093,E2 -20559.093} C_VEL
LIN {X 0,Y 225.343,Z 329.818,A -85,B 0,C 180,E1 -20560.023,E2 -20560.023} C_VEL
LIN {X 0,Y 227.223,Z 333.355,A -85,B 0,C 180,E1 -20560.798,E2 -20560.798} C_VEL
LIN {X 0,Y 228.538,Z 335.247,A -85,B 0,C 180,E1 -20561.315,E2 -20561.315} C_VEL
LIN {X 0,Y 230.756,Z 339.184,A -85,B 0,C 180,E1 -20562.217,E2 -20562.217} C_VEL
LIN {X 0,Y 235.178,Z 348.414,A -85,B 0,C 180,E1 -20564.151,E2 -20564.151} C_VEL
LIN {X 0,Y 238.937,Z 358.669,A -85,B 0,C 180,E1 -20566.105,E2 -20566.105} C_VEL
LIN {X 0,Y 242.295,Z 371.013,A -85,B 0,C 180,E1 -20568.323,E2 -20568.323} C_VEL
LIN {X 0,Y 243.089,Z 374.88,A -85,B 0,C 180,E1 -20569.021,E2 -20569.021} C_VEL
LIN {X 0,Y 243.414,Z 379.816,A -85,B 0,C 180,E1 -20569.789,E2 -20569.789} C_VEL
LIN {X 0,Y 242.036,Z 388.477,A -85,B 0,C 180,E1 -20570.902,E2 -20570.902} C_VEL
LIN {X 0,Y 239.847,Z 398.669,A -85,B 0,C 180,E1 -20572.329,E2 -20572.329} C_VEL
LIN {X 0,Y 239.564,Z 401.756,A -85,B 0,C 180,E1 -20572.904,E2 -20572.904} C_VEL
LIN {X 0,Y 237.965,Z 407.335,A -85,B 0,C 180,E1 -20573.795,E2 -20573.795} C_VEL
LIN {X 0,Y 234.096,Z 418.357,A -85,B 0,C 180,E1 -20575.743,E2 -20575.743} C_VEL
LIN {X 0,Y 229.887,Z 429.495,A -85,B 0,C 180,E1 -20578.173,E2 -20578.173} C_VEL
LIN {X 0,Y 226.121,Z 438.705,A -85,B 0,C 180,E1 -20580.635,E2 -20580.635} C_VEL
LIN {X 0,Y 222.865,Z 446.853,A -85,B 0,C 180,E1 -20583.296,E2 -20583.296} C_VEL
LIN {X 0,Y 219.457,Z 454.743,A -85,B 0,C 180,E1 -20586.402,E2 -20586.402} C_VEL
LIN {X 0,Y 216.348,Z 462.111,A -85,B 0,C 180,E1 -20590.057,E2 -20590.057} C_VEL
LIN {X 0,Y 214.163,Z 467.954,A -85,B 0,C 180,E1 -20593.803,E2 -20593.803} C_VEL
LIN {X 0,Y 212.875,Z 471.429,A -85,B 0,C 180,E1 -20596.637,E2 -20596.637} C_VEL
LIN {X 0,Y 211.886,Z 474.939,A -85,B 0,C 180,E1 -20600.453,E2 -20600.453} C_VEL
LIN {X 0,Y 211.405,Z 477.247,A -85,B 0,C 180,E1 -20604.276,E2 -20604.276} C_VEL
LIN {X 0,Y 211.353,Z 478.407,A -85,B 0,C 180,E1 -20608.094,E2 -20608.094} C_VEL
LIN {X 0,Y 211.431,Z 478.56,A -85,B 0,C 180,E1 -20609.999,E2 -20609.999} C_VEL
LIN {X 0,Y 211.335,Z 477.927,A -85,B 0,C 180,E1 -20613.926,E2 -20613.926} C_VEL
LIN {X 0,Y 211.596,Z 476.209,A -85,B 0,C 180,E1 -20617.634,E2 -20617.634} C_VEL
LIN {X 0,Y 212.297,Z 473.295,A -85,B 0,C 180,E1 -20621.456,E2 -20621.456} C_VEL
LIN {X 0,Y 213.705,Z 469.146,A -85,B 0,C 180,E1 -20625.253,E2 -20625.253} C_VEL
LIN {X 0,Y 215.904,Z 463.204,A -85,B 0,C 180,E1 -20629.268,E2 -20629.268} C_VEL
LIN {X 0,Y 218.599,Z 456.661,A -85,B 0,C 180,E1 -20632.692,E2 -20632.692} C_VEL
LIN {X 0,Y 222.303,Z 447.964,A -85,B 0,C 180,E1 -20636.269,E2 -20636.269} C_VEL
LIN {X 0,Y 225.954,Z 439.184,A -85,B 0,C 180,E1 -20639.174,E2 -20639.174} C_VEL
LIN {X 0,Y 229.877,Z 429.331,A -85,B 0,C 180,E1 -20641.827,E2 -20641.827} C_VEL
LIN {X 0,Y 234.455,Z 417.142,A -85,B 0,C 180,E1 -20644.456,E2 -20644.456} C_VEL
LIN {X 0,Y 238.455,Z 405.686,A -85,B 0,C 180,E1 -20646.435,E2 -20646.435} C_VEL
LIN {X 0,Y 239.435,Z 402.347,A -85,B 0,C 180,E1 -20646.946,E2 -20646.946} C_VEL
LIN {X 0,Y 239.099,Z 391.655,A -85,B 0,C 180,E1 -20649.064,E2 -20649.064} C_VEL
LIN {X 0,Y 237.55,Z 378.744,A -85,B 0,C 180,E1 -20651.512,E2 -20651.512} C_VEL
LIN {X 0,Y 234.62,Z 365.372,A -85,B 0,C 180,E1 -20654.035,E2 -20654.035} C_VEL
LIN {X 0,Y 230.574,Z 353.078,A -85,B 0,C 180,E1 -20656.476,E2 -20656.476} C_VEL
LIN {X 0,Y 226.67,Z 344.307,A -85,B 0,C 180,E1 -20658.402,E2 -20658.402} C_VEL
LIN {X 0,Y 223.6,Z 338.893,A -85,B 0,C 180,E1 -20659.776,E2 -20659.776} C_VEL
LIN {X 0,Y 220.981,Z 334.323,A -85,B 0,C 180,E1 -20660.942,E2 -20660.942} C_VEL
LIN {X 0,Y 218.641,Z 330.695,A -85,B 0,C 180,E1 -20661.962,E2 -20661.962} C_VEL
LIN {X 0,Y 217.891,Z 329.184,A -85,B 0,C 180,E1 -20662.308,E2 -20662.308} C_VEL
LIN {X 0,Y 215.603,Z 326.43,A -85,B 0,C 180,E1 -20663.277,E2 -20663.277} C_VEL
LIN {X 0,Y 214.528,Z 323.548,A -85,B 0,C 180,E1 -20663.866,E2 -20663.866} C_VEL
LIN {X 0,Y 214.18,Z 321.189,A -85,B 0,C 180,E1 -20668.553,E2 -20668.553} C_VEL
LIN {X 0,Y 213.929,Z 319.366,A -85,B 0,C 180,E1 -20672.618,E2 -20672.618} C_VEL
LIN {X 0,Y 213.801,Z 318.516,A -85,B 0,C 180,E1 -20674.702,E2 -20674.702} C_VEL
LIN {X 0,Y 213.808,Z 318.477,A -85,B 0,C 180,E1 -20678.803,E2 -20678.803} C_VEL
LIN {X 0,Y 213.938,Z 318.457,A -85,B 0,C 180,E1 -20682.803,E2 -20682.803} C_VEL
LIN {X 0,Y 213.944,Z 318.461,A -85,B 0,C 180,E1 -20686.706,E2 -20686.706} C_VEL
LIN {X 0,Y 214.127,Z 318.433,A -85,B 0,C 180,E1 -20690.555,E2 -20690.555} C_VEL
LIN {X 0,Y 214.082,Z 318.437,A -85,B 0,C 180,E1 -20694.348,E2 -20694.348} C_VEL
LIN {X 0,Y 214.438,Z 318.392,A -85,B 0,C 180,E1 -20698.122,E2 -20698.122} C_VEL
LIN {X 0,Y 214.536,Z 318.387,A -85,B 0,C 180,E1 -20700,E2 -20700} C_VEL
LIN {X 0,Y 214.438,Z 318.398,A -85,B 0,C 180,E1 -20701.878,E2 -20701.878} C_VEL
LIN {X 0,Y 214.175,Z 318.427,A -85,B 0,C 180,E1 -20707.542,E2 -20707.542} C_VEL
LIN {X 0,Y 213.992,Z 318.449,A -85,B 0,C 180,E1 -20711.365,E2 -20711.365} C_VEL
LIN {X 0,Y 213.926,Z 318.458,A -85,B 0,C 180,E1 -20715.238,E2 -20715.238} C_VEL
LIN {X 0,Y 213.864,Z 318.471,A -85,B 0,C 180,E1 -20719.185,E2 -20719.185} C_VEL
LIN {X 0,Y 213.843,Z 318.473,A -85,B 0,C 180,E1 -20723.228,E2 -20723.228} C_VEL
LIN {X 0,Y 213.825,Z 318.472,A -85,B 0,C 180,E1 -20727.451,E2 -20727.451} C_VEL
LIN {X 0,Y 213.756,Z 318.488,A -85,B 0,C 180,E1 -20729.55,E2 -20729.55} C_VEL
LIN {X 0,Y 214.059,Z 320.271,A -85,B 0,C 180,E1 -20733.928,E2 -20733.928} C_VEL
LIN {X 0,Y 214.197,Z 321.363,A -85,B 0,C 180,E1 -20736.1,E2 -20736.1} C_VEL
LIN {X 0,Y 215.23,Z 324.019,A -85,B 0,C 180,E1 -20736.641,E2 -20736.641} C_VEL
LIN {X 0,Y 217.558,Z 326.75,A -85,B 0,C 180,E1 -20737.633,E2 -20737.633} C_VEL
LIN {X 0,Y 220.137,Z 331.171,A -85,B 0,C 180,E1 -20738.795,E2 -20738.795} C_VEL
LIN {X 0,Y 221.406,Z 332.842,A -85,B 0,C 180,E1 -20739.336,E2 -20739.336} C_VEL
LIN {X 0,Y 223.795,Z 336.862,A -85,B 0,C 180,E1 -20740.387,E2 -20740.387} C_VEL
LIN {X 0,Y 228.728,Z 346.255,A -85,B 0,C 180,E1 -20742.68,E2 -20742.68} C_VEL
LIN {X 0,Y 232.733,Z 355.998,A -85,B 0,C 180,E1 -20744.8,E2 -20744.8} C_VEL
LIN {X 0,Y 235.927,Z 366.323,A -85,B 0,C 180,E1 -20746.871,E2 -20746.871} C_VEL
LIN {X 0,Y 238.371,Z 377.499,A -85,B 0,C 180,E1 -20749.062,E2 -20749.062} C_VEL
LIN {X 0,Y 239.963,Z 388.608,A -85,B 0,C 180,E1 -20751.252,E2 -20751.252} C_VEL
LIN {X 0,Y 240.46,Z 396.653,A -85,B 0,C 180,E1 -20752.882,E2 -20752.882} C_VEL
LIN {X 0,Y 236.531,Z 408.924,A -85,B 0,C 180,E1 -20754.854,E2 -20754.854} C_VEL
LIN {X 0,Y 232.525,Z 420.048,A -85,B 0,C 180,E1 -20757.042,E2 -20757.042} C_VEL
LIN {X 0,Y 228.423,Z 430.677,A -85,B 0,C 180,E1 -20759.626,E2 -20759.626} C_VEL
LIN {X 0,Y 224.466,Z 440.251,A -85,B 0,C 180,E1 -20762.497,E2 -20762.497} C_VEL
LIN {X 0,Y 220.919,Z 448.537,A -85,B 0,C 180,E1 -20765.572,E2 -20765.572} C_VEL
LIN {X 0,Y 217.606,Z 456.322,A -85,B 0,C 180,E1 -20769.191,E2 -20769.191} C_VEL
LIN {X 0,Y 215.092,Z 462.517,A -85,B 0,C 180,E1 -20772.899,E2 -20772.899} C_VEL
LIN {X 0,Y 213.204,Z 467.3,A -85,B 0,C 180,E1 -20776.66,E2 -20776.66} C_VEL
LIN {X 0,Y 212.094,Z 470.802,A -85,B 0,C 180,E1 -20780.464,E2 -20780.464} C_VEL
LIN {X 0,Y 211.514,Z 473.115,A -85,B 0,C 180,E1 -20784.28,E2 -20784.28} C_VEL
LIN {X 0,Y 211.395,Z 474.291,A -85,B 0,C 180,E1 -20788.096,E2 -20788.096} C_VEL
LIN {X 0,Y 211.438,Z 474.448,A -85,B 0,C 180,E1 -20790.001,E2 -20790.001} C_VEL
LIN {X 0,Y 211.42,Z 473.772,A -85,B 0,C 180,E1 -20794.242,E2 -20794.242} C_VEL
LIN {X 0,Y 211.725,Z 472.186,A -85,B 0,C 180,E1 -20797.631,E2 -20797.631} C_VEL
LIN {X 0,Y 212.581,Z 469.331,A -85,B 0,C 180,E1 -20801.442,E2 -20801.442} C_VEL
LIN {X 0,Y 214.035,Z 465.245,A -85,B 0,C 180,E1 -20805.23,E2 -20805.23} C_VEL
LIN {X 0,Y 216.183,Z 459.828,A -85,B 0,C 180,E1 -20808.972,E2 -20808.972} C_VEL
LIN {X 0,Y 219.056,Z 452.927,A -85,B 0,C 180,E1 -20812.644,E2 -20812.644} C_VEL
LIN {X 0,Y 222.738,Z 444.315,A -85,B 0,C 180,E1 -20816.215,E2 -20816.215} C_VEL
LIN {X 0,Y 226.726,Z 435.157,A -85,B 0,C 180,E1 -20819.224,E2 -20819.224} C_VEL
LIN {X 0,Y 230.379,Z 425.834,A -85,B 0,C 180,E1 -20821.751,E2 -20821.751} C_VEL
LIN {X 0,Y 234.914,Z 413.765,A -85,B 0,C 180,E1 -20824.381,E2 -20824.381} C_VEL
LIN {X 0,Y 239.303,Z 400.952,A -85,B 0,C 180,E1 -20826.593,E2 -20826.593} C_VEL
LIN {X 0,Y 240.495,Z 397.122,A -85,B 0,C 180,E1 -20827.158,E2 -20827.158} C_VEL
LIN {X 0,Y 239.669,Z 385.654,A -85,B 0,C 180,E1 -20829.467,E2 -20829.467} C_VEL
LIN {X 0,Y 237.995,Z 374.936,A -85,B 0,C 180,E1 -20831.58,E2 -20831.58} C_VEL
LIN {X 0,Y 235.147,Z 363.323,A -85,B 0,C 180,E1 -20833.859,E2 -20833.859} C_VEL
LIN {X 0,Y 231.191,Z 351.787,A -85,B 0,C 180,E1 -20836.245,E2 -20836.245} C_VEL
LIN {X 0,Y 227.619,Z 343.972,A -85,B 0,C 180,E1 -20838.021,E2 -20838.021} C_VEL
LIN {X 0,Y 223.383,Z 336.308,A -85,B 0,C 180,E1 -20839.956,E2 -20839.956} C_VEL
LIN {X 0,Y 220.661,Z 331.778,A -85,B 0,C 180,E1 -20841.168,E2 -20841.168} C_VEL
LIN {X 0,Y 218.435,Z 328.457,A -85,B 0,C 180,E1 -20842.148,E2 -20842.148} C_VEL
LIN {X 0,Y 217.496,Z 326.692,A -85,B 0,C 180,E1 -20842.58,E2 -20842.58} C_VEL
LIN {X 0,Y 215.115,Z 323.865,A -85,B 0,C 180,E1 -20843.604,E2 -20843.604} C_VEL
LIN {X 0,Y 214.188,Z 321.214,A -85,B 0,C 180,E1 -20844.191,E2 -20844.191} C_VEL
LIN {X 0,Y 213.877,Z 319.274,A -85,B 0,C 180,E1 -20848.689,E2 -20848.689} C_VEL
LIN {X 0,Y 213.752,Z 318.588,A -85,B 0,C 180,E1 -20850.449,E2 -20850.449} C_VEL
LIN {X 0,Y 213.782,Z 318.48,A -85,B 0,C 180,E1 -20854.699,E2 -20854.699} C_VEL
LIN {X 0,Y 213.806,Z 318.476,A -85,B 0,C 180,E1 -20858.802,E2 -20858.802} C_VEL
LIN {X 0,Y 213.944,Z 318.458,A -85,B 0,C 180,E1 -20862.803,E2 -20862.803} C_VEL
LIN {X 0,Y 213.946,Z 318.453,A -85,B 0,C 180,E1 -20866.706,E2 -20866.706} C_VEL
LIN {X 0,Y 214.134,Z 318.438,A -85,B 0,C 180,E1 -20870.555,E2 -20870.555} C_VEL
LIN {X 0,Y 214.087,Z 318.444,A -85,B 0,C 180,E1 -20874.348,E2 -20874.348} C_VEL
LIN {X 0,Y 214.443,Z 318.398,A -85,B 0,C 180,E1 -20878.122,E2 -20878.122} C_VEL
LIN {X 0,Y 214.538,Z 318.386,A -85,B 0,C 180,E1 -20880,E2 -20880} C_VEL
LIN {X 0,Y 214.443,Z 318.399,A -85,B 0,C 180,E1 -20881.878,E2 -20881.878} C_VEL
LIN {X 0,Y 214.185,Z 318.431,A -85,B 0,C 180,E1 -20887.542,E2 -20887.542} C_VEL
LIN {X 0,Y 213.999,Z 318.455,A -85,B 0,C 180,E1 -20891.364,E2 -20891.364} C_VEL
LIN {X 0,Y 213.933,Z 318.464,A -85,B 0,C 180,E1 -20895.237,E2 -20895.237} C_VEL
LIN {X 0,Y 213.835,Z 318.474,A -85,B 0,C 180,E1 -20899.187,E2 -20899.187} C_VEL
LIN {X 0,Y 213.811,Z 318.478,A -85,B 0,C 180,E1 -20903.231,E2 -20903.231} C_VEL
LIN {X 0,Y 213.827,Z 318.566,A -85,B 0,C 180,E1 -20905.295,E2 -20905.295} C_VEL
LIN {X 0,Y 214.047,Z 320.348,A -85,B 0,C 180,E1 -20909.505,E2 -20909.505} C_VEL
LIN {X 0,Y 214.355,Z 322.427,A -85,B 0,C 180,E1 -20913.874,E2 -20913.874} C_VEL
LIN {X 0,Y 214.511,Z 323.561,A -85,B 0,C 180,E1 -20916.052,E2 -20916.052} C_VEL
LIN {X 0,Y 215.536,Z 326.318,A -85,B 0,C 180,E1 -20916.591,E2 -20916.591} C_VEL
LIN {X 0,Y 217.877,Z 329.196,A -85,B 0,C 180,E1 -20917.591,E2 -20917.591} C_VEL
LIN {X 0,Y 220.424,Z 333.643,A -85,B 0,C 180,E1 -20918.735,E2 -20918.735} C_VEL
LIN {X 0,Y 221.794,Z 335.6,A -85,B 0,C 180,E1 -20919.326,E2 -20919.326} C_VEL
LIN {X 0,Y 224.28,Z 339.769,A -85,B 0,C 180,E1 -20920.41,E2 -20920.41} C_VEL
LIN {X 0,Y 228.796,Z 348.665,A -85,B 0,C 180,E1 -20922.515,E2 -20922.515} C_VEL
LIN {X 0,Y 232.42,Z 358.034,A -85,B 0,C 180,E1 -20924.473,E2 -20924.473} C_VEL
LIN {X 0,Y 235.327,Z 367.971,A -85,B 0,C 180,E1 -20926.404,E2 -20926.404} C_VEL
LIN {X 0,Y 237.866,Z 380.235,A -85,B 0,C 180,E1 -20928.73,E2 -20928.73} C_VEL
LIN {X 0,Y 239.192,Z 391.674,A -85,B 0,C 180,E1 -20930.9,E2 -20930.9} C_VEL
LIN {X 0,Y 239.564,Z 401.756,A -85,B 0,C 180,E1 -20932.904,E2 -20932.904} C_VEL
LIN {X 0,Y 238.986,Z 404.922,A -85,B 0,C 180,E1 -20933.444,E2 -20933.444} C_VEL
LIN {X 0,Y 236.734,Z 409.587,A -85,B 0,C 180,E1 -20934.079,E2 -20934.079} C_VEL
LIN {X 0,Y 227.755,Z 421.621,A -85,B 0,C 180,E1 -20935.558,E2 -20935.558} C_VEL
LIN {X 0,Y 225.251,Z 425.973,A -85,B 0,C 180,E1 -20936.397,E2 -20936.397} C_VEL
LIN {X 0,Y 221.118,Z 435.824,A -85,B 0,C 180,E1 -20938.903,E2 -20938.903} C_VEL
LIN {X 0,Y 217.047,Z 445.551,A -85,B 0,C 180,E1 -20941.997,E2 -20941.997} C_VEL
LIN {X 0,Y 213.378,Z 453.664,A -85,B 0,C 180,E1 -20945.168,E2 -20945.168} C_VEL
LIN {X 0,Y 210.354,Z 460.374,A -85,B 0,C 180,E1 -20948.437,E2 -20948.437} C_VEL
LIN {X 0,Y 207.79,Z 466.569,A -85,B 0,C 180,E1 -20952.277,E2 -20952.277} C_VEL
LIN {X 0,Y 205.922,Z 471.36,A -85,B 0,C 180,E1 -20956.177,E2 -20956.177} C_VEL
LIN {X 0,Y 204.85,Z 474.87,A -85,B 0,C 180,E1 -20960.122,E2 -20960.122} C_VEL
LIN {X 0,Y 204.337,Z 477.179,A -85,B 0,C 180,E1 -20964.077,E2 -20964.077} C_VEL
LIN {X 0,Y 204.261,Z 478.339,A -85,B 0,C 180,E1 -20968.028,E2 -20968.028} C_VEL
LIN {X 0,Y 204.334,Z 478.491,A -85,B 0,C 180,E1 -20969.999,E2 -20969.999} C_VEL
LIN {X 0,Y 204.256,Z 477.886,A -85,B 0,C 180,E1 -20973.945,E2 -20973.945} C_VEL
LIN {X 0,Y 204.534,Z 476.139,A -85,B 0,C 180,E1 -20977.899,E2 -20977.899} C_VEL
LIN {X 0,Y 205.306,Z 473.225,A -85,B 0,C 180,E1 -20981.851,E2 -20981.851} C_VEL
LIN {X 0,Y 206.814,Z 469.076,A -85,B 0,C 180,E1 -20985.774,E2 -20985.774} C_VEL
LIN {X 0,Y 209.015,Z 463.498,A -85,B 0,C 180,E1 -20989.699,E2 -20989.699} C_VEL
LIN {X 0,Y 212.011,Z 456.589,A -85,B 0,C 180,E1 -20993.439,E2 -20993.439} C_VEL
LIN {X 0,Y 215.94,Z 447.893,A -85,B 0,C 180,E1 -20997.105,E2 -20997.105} C_VEL
LIN {X 0,Y 219.953,Z 438.603,A -85,B 0,C 180,E1 -21000.231,E2 -21000.231} C_VEL
LIN {X 0,Y 223.838,Z 429.259,A -85,B 0,C 180,E1 -21002.792,E2 -21002.792} C_VEL
LIN {X 0,Y 228.628,Z 417.07,A -85,B 0,C 180,E1 -21005.464,E2 -21005.464} C_VEL
LIN {X 0,Y 233.03,Z 404.749,A -85,B 0,C 180,E1 -21007.617,E2 -21007.617} C_VEL
LIN {X 0,Y 233.317,Z 401.904,A -85,B 0,C 180,E1 -21008.162,E2 -21008.162} C_VEL
LIN {X 0,Y 232.932,Z 391.499,A -85,B 0,C 180,E1 -21010.319,E2 -21010.319} C_VEL
LIN {X 0,Y 231.812,Z 381.193,A -85,B 0,C 180,E1 -21012.359,E2 -21012.359} C_VEL
LIN {X 0,Y 229.378,Z 369.021,A -85,B 0,C 180,E1 -21014.804,E2 -21014.804} C_VEL
LIN {X 0,Y 225.652,Z 356.716,A -85,B 0,C 180,E1 -21017.385,E2 -21017.385} C_VEL
LIN {X 0,Y 221.938,Z 348.362,A -85,B 0,C 180,E1 -21019.395,E2 -21019.395} C_VEL
LIN {X 0,Y 218.951,Z 342.845,A -85,B 0,C 180,E1 -21020.862,E2 -21020.862} C_VEL
LIN {X 0,Y 217.283,Z 339.697,A -85,B 0,C 180,E1 -21021.713,E2 -21021.713} C_VEL
LIN {X 0,Y 214.825,Z 335.498,A -85,B 0,C 180,E1 -21022.902,E2 -21022.902} C_VEL
LIN {X 0,Y 211.906,Z 331.129,A -85,B 0,C 180,E1 -21024.315,E2 -21024.315} C_VEL
LIN {X 0,Y 210.872,Z 329.189,A -85,B 0,C 180,E1 -21024.84,E2 -21024.84} C_VEL
LIN {X 0,Y 208.567,Z 326.599,A -85,B 0,C 180,E1 -21025.93,E2 -21025.93} C_VEL
LIN {X 0,Y 207.415,Z 323.866,A -85,B 0,C 180,E1 -21026.591,E2 -21026.591} C_VEL
LIN {X 0,Y 207.313,Z 323.426,A -85,B 0,C 180,E1 -21026.718,E2 -21026.718} C_VEL
LIN {X 0,Y 206.997,Z 321.21,A -85,B 0,C 180,E1 -21031.619,E2 -21031.619} C_VEL
LIN {X 0,Y 206.781,Z 319.352,A -85,B 0,C 180,E1 -21036.584,E2 -21036.584} C_VEL
LIN {X 0,Y 206.868,Z 319.339,A -85,B 0,C 180,E1 -21042.196,E2 -21042.196} C_VEL
LIN {X 0,Y 206.887,Z 319.339,A -85,B 0,C 180,E1 -21046.244,E2 -21046.244} C_VEL
LIN {X 0,Y 207.072,Z 319.314,A -85,B 0,C 180,E1 -21050.23,E2 -21050.23} C_VEL
LIN {X 0,Y 207.043,Z 319.314,A -85,B 0,C 180,E1 -21054.155,E2 -21054.155} C_VEL
LIN {X 0,Y 207.374,Z 319.272,A -85,B 0,C 180,E1 -21058.058,E2 -21058.058} C_VEL
LIN {X 0,Y 207.502,Z 319.263,A -85,B 0,C 180,E1 -21060,E2 -21060} C_VEL
LIN {X 0,Y 207.374,Z 319.278,A -85,B 0,C 180,E1 -21061.942,E2 -21061.942} C_VEL
LIN {X 0,Y 207.12,Z 319.304,A -85,B 0,C 180,E1 -21067.801,E2 -21067.801} C_VEL
LIN {X 0,Y 206.917,Z 319.33,A -85,B 0,C 180,E1 -21071.759,E2 -21071.759} C_VEL
LIN {X 0,Y 206.86,Z 319.341,A -85,B 0,C 180,E1 -21075.771,E2 -21075.771} C_VEL
LIN {X 0,Y 206.795,Z 319.348,A -85,B 0,C 180,E1 -21079.868,E2 -21079.868} C_VEL
LIN {X 0,Y 206.759,Z 319.356,A -85,B 0,C 180,E1 -21084.073,E2 -21084.073} C_VEL
LIN {X 0,Y 206.733,Z 319.498,A -85,B 0,C 180,E1 -21088.421,E2 -21088.421} C_VEL
LIN {X 0,Y 207.01,Z 321.356,A -85,B 0,C 180,E1 -21093.265,E2 -21093.265} C_VEL
LIN {X 0,Y 208.138,Z 324.214,A -85,B 0,C 180,E1 -21093.931,E2 -21093.931} C_VEL
LIN {X 0,Y 210.44,Z 326.888,A -85,B 0,C 180,E1 -21095.042,E2 -21095.042} C_VEL
LIN {X 0,Y 211.127,Z 327.818,A -85,B 0,C 180,E1 -21095.371,E2 -21095.371} C_VEL
LIN {X 0,Y 213.064,Z 331.159,A -85,B 0,C 180,E1 -21096.351,E2 -21096.351} C_VEL
LIN {X 0,Y 214.606,Z 333.253,A -85,B 0,C 180,E1 -21097.089,E2 -21097.089} C_VEL
LIN {X 0,Y 216.968,Z 337.148,A -85,B 0,C 180,E1 -21098.232,E2 -21098.232} C_VEL
LIN {X 0,Y 218.271,Z 339.477,A -85,B 0,C 180,E1 -21098.894,E2 -21098.894} C_VEL
LIN {X 0,Y 222.624,Z 347.427,A -85,B 0,C 180,E1 -21101.069,E2 -21101.069} C_VEL
LIN {X 0,Y 226.284,Z 355.856,A -85,B 0,C 180,E1 -21103.101,E2 -21103.101} C_VEL
LIN {X 0,Y 229.891,Z 366.976,A -85,B 0,C 180,E1 -21105.522,E2 -21105.522} C_VEL
LIN {X 0,Y 232.583,Z 379.576,A -85,B 0,C 180,E1 -21108.145,E2 -21108.145} C_VEL
LIN {X 0,Y 234.027,Z 391.488,A -85,B 0,C 180,E1 -21110.626,E2 -21110.626} C_VEL
LIN {X 0,Y 234.326,Z 398.042,A -85,B 0,C 180,E1 -21112.017,E2 -21112.017} C_VEL
LIN {X 0,Y 230.36,Z 410.063,A -85,B 0,C 180,E1 -21114.036,E2 -21114.036} C_VEL
LIN {X 0,Y 225.855,Z 421.9,A -85,B 0,C 180,E1 -21116.474,E2 -21116.474} C_VEL
LIN {X 0,Y 221.653,Z 432.332,A -85,B 0,C 180,E1 -21119.157,E2 -21119.157} C_VEL
LIN {X 0,Y 217.562,Z 441.589,A -85,B 0,C 180,E1 -21122.071,E2 -21122.071} C_VEL
LIN {X 0,Y 213.929,Z 449.699,A -85,B 0,C 180,E1 -21125.238,E2 -21125.238} C_VEL
LIN {X 0,Y 210.919,Z 456.393,A -85,B 0,C 180,E1 -21128.499,E2 -21128.499} C_VEL
LIN {X 0,Y 208.247,Z 462.588,A -85,B 0,C 180,E1 -21132.319,E2 -21132.319} C_VEL
LIN {X 0,Y 206.252,Z 467.371,A -85,B 0,C 180,E1 -21136.202,E2 -21136.202} C_VEL
LIN {X 0,Y 205.079,Z 470.872,A -85,B 0,C 180,E1 -21140.135,E2 -21140.135} C_VEL
LIN {X 0,Y 204.444,Z 473.184,A -85,B 0,C 180,E1 -21144.082,E2 -21144.082} C_VEL
LIN {X 0,Y 204.303,Z 474.36,A -85,B 0,C 180,E1 -21148.029,E2 -21148.029} C_VEL
LIN {X 0,Y 204.342,Z 474.517,A -85,B 0,C 180,E1 -21150.001,E2 -21150.001} C_VEL
LIN {X 0,Y 204.322,Z 473.924,A -85,B 0,C 180,E1 -21154.045,E2 -21154.045} C_VEL
LIN {X 0,Y 204.669,Z 472.255,A -85,B 0,C 180,E1 -21157.895,E2 -21157.895} C_VEL
LIN {X 0,Y 205.573,Z 469.4,A -85,B 0,C 180,E1 -21161.837,E2 -21161.837} C_VEL
LIN {X 0,Y 207.166,Z 465.313,A -85,B 0,C 180,E1 -21165.748,E2 -21165.748} C_VEL
LIN {X 0,Y 209.436,Z 459.896,A -85,B 0,C 180,E1 -21169.608,E2 -21169.608} C_VEL
LIN {X 0,Y 212.489,Z 452.995,A -85,B 0,C 180,E1 -21173.385,E2 -21173.385} C_VEL
LIN {X 0,Y 216.34,Z 444.382,A -85,B 0,C 180,E1 -21177.053,E2 -21177.053} C_VEL
LIN {X 0,Y 220.516,Z 435.224,A -85,B 0,C 180,E1 -21180.13,E2 -21180.13} C_VEL
LIN {X 0,Y 224.347,Z 425.901,A -85,B 0,C 180,E1 -21182.71,E2 -21182.71} C_VEL
LIN {X 0,Y 229.047,Z 413.831,A -85,B 0,C 180,E1 -21185.391,E2 -21185.391} C_VEL
LIN {X 0,Y 233.201,Z 402.295,A -85,B 0,C 180,E1 -21187.43,E2 -21187.43} C_VEL
LIN {X 0,Y 234.395,Z 398.547,A -85,B 0,C 180,E1 -21188.009,E2 -21188.009} C_VEL
LIN {X 0,Y 233.621,Z 386.585,A -85,B 0,C 180,E1 -21190.544,E2 -21190.544} C_VEL
LIN {X 0,Y 232.11,Z 376.603,A -85,B 0,C 180,E1 -21192.614,E2 -21192.614} C_VEL
LIN {X 0,Y 229.524,Z 365.572,A -85,B 0,C 180,E1 -21194.923,E2 -21194.923} C_VEL
LIN {X 0,Y 226.5,Z 356.304,A -85,B 0,C 180,E1 -21196.95,E2 -21196.95} C_VEL
LIN {X 0,Y 222.245,Z 346.542,A -85,B 0,C 180,E1 -21199.318,E2 -21199.318} C_VEL
LIN {X 0,Y 217.165,Z 337.374,A -85,B 0,C 180,E1 -21201.867,E2 -21201.867} C_VEL
LIN {X 0,Y 214.8,Z 333.629,A -85,B 0,C 180,E1 -21203.001,E2 -21203.001} C_VEL
LIN {X 0,Y 213.789,Z 332.004,A -85,B 0,C 180,E1 -21203.504,E2 -21203.504} C_VEL
LIN {X 0,Y 211.547,Z 328.756,A -85,B 0,C 180,E1 -21204.603,E2 -21204.603} C_VEL
LIN {X 0,Y 210.627,Z 327.021,A -85,B 0,C 180,E1 -21205.078,E2 -21205.078} C_VEL
LIN {X 0,Y 208.328,Z 324.511,A -85,B 0,C 180,E1 -21206.177,E2 -21206.177} C_VEL
LIN {X 0,Y 207.086,Z 321.68,A -85,B 0,C 180,E1 -21206.894,E2 -21206.894} C_VEL
LIN {X 0,Y 206.989,Z 321.305,A -85,B 0,C 180,E1 -21207.094,E2 -21207.094} C_VEL
LIN {X 0,Y 206.738,Z 319.4,A -85,B 0,C 180,E1 -21212.112,E2 -21212.112} C_VEL
LIN {X 0,Y 206.746,Z 319.358,A -85,B 0,C 180,E1 -21216.61,E2 -21216.61} C_VEL
LIN {X 0,Y 206.874,Z 319.342,A -85,B 0,C 180,E1 -21222.196,E2 -21222.196} C_VEL
LIN {X 0,Y 206.89,Z 319.335,A -85,B 0,C 180,E1 -21226.244,E2 -21226.244} C_VEL
LIN {X 0,Y 207.078,Z 319.315,A -85,B 0,C 180,E1 -21230.23,E2 -21230.23} C_VEL
LIN {X 0,Y 207.048,Z 319.32,A -85,B 0,C 180,E1 -21234.155,E2 -21234.155} C_VEL
LIN {X 0,Y 207.379,Z 319.278,A -85,B 0,C 180,E1 -21238.058,E2 -21238.058} C_VEL
LIN {X 0,Y 207.504,Z 319.262,A -85,B 0,C 180,E1 -21240,E2 -21240} C_VEL
LIN {X 0,Y 207.379,Z 319.279,A -85,B 0,C 180,E1 -21241.942,E2 -21241.942} C_VEL
LIN {X 0,Y 207.129,Z 319.311,A -85,B 0,C 180,E1 -21247.8,E2 -21247.8} C_VEL
LIN {X 0,Y 206.924,Z 319.337,A -85,B 0,C 180,E1 -21251.758,E2 -21251.758} C_VEL
LIN {X 0,Y 206.867,Z 319.342,A -85,B 0,C 180,E1 -21255.771,E2 -21255.771} C_VEL
LIN {X 0,Y 206.778,Z 319.354,A -85,B 0,C 180,E1 -21259.869,E2 -21259.869} C_VEL
LIN {X 0,Y 206.79,Z 319.568,A -85,B 0,C 180,E1 -21264.069,E2 -21264.069} C_VEL
LIN {X 0,Y 207.005,Z 321.259,A -85,B 0,C 180,E1 -21268.379,E2 -21268.379} C_VEL
LIN {X 0,Y 207.31,Z 323.446,A -85,B 0,C 180,E1 -21273.21,E2 -21273.21} C_VEL
LIN {X 0,Y 208.424,Z 326.355,A -85,B 0,C 180,E1 -21273.878,E2 -21273.878} C_VEL
LIN {X 0,Y 210.806,Z 329.154,A -85,B 0,C 180,E1 -21275.022,E2 -21275.022} C_VEL
LIN {X 0,Y 211.356,Z 329.897,A -85,B 0,C 180,E1 -21275.284,E2 -21275.284} C_VEL
LIN {X 0,Y 213.233,Z 333.349,A -85,B 0,C 180,E1 -21276.241,E2 -21276.241} C_VEL
LIN {X 0,Y 214.864,Z 335.551,A -85,B 0,C 180,E1 -21277.017,E2 -21277.017} C_VEL
LIN {X 0,Y 217.316,Z 339.725,A -85,B 0,C 180,E1 -21278.207,E2 -21278.207} C_VEL
LIN {X 0,Y 221.111,Z 346.776,A -85,B 0,C 180,E1 -21280.11,E2 -21280.11} C_VEL
LIN {X 0,Y 224.236,Z 353.127,A -85,B 0,C 180,E1 -21281.729,E2 -21281.729} C_VEL
LIN {X 0,Y 227.866,Z 363.245,A -85,B 0,C 180,E1 -21283.944,E2 -21283.944} C_VEL
LIN {X 0,Y 230.486,Z 373.703,A -85,B 0,C 180,E1 -21286.084,E2 -21286.084} C_VEL
LIN {X 0,Y 232.39,Z 384.77,A -85,B 0,C 180,E1 -21288.292,E2 -21288.292} C_VEL
LIN {X 0,Y 233.349,Z 396.955,A -85,B 0,C 180,E1 -21290.767,E2 -21290.767} C_VEL
LIN {X 0,Y 233.437,Z 403.646,A -85,B 0,C 180,E1 -21292.172,E2 -21292.172} C_VEL
LIN {X 0,Y 229.033,Z 416.212,A -85,B 0,C 180,E1 -21294.336,E2 -21294.336} C_VEL
LIN {X 0,Y 225.251,Z 425.973,A -85,B 0,C 180,E1 -21296.397,E2 -21296.397} C_VEL
LIN {X 0,Y 223.512,Z 428.817,A -85,B 0,C 180,E1 -21296.963,E2 -21296.963} C_VEL
LIN {X 0,Y 214.85,Z 437.448,A -85,B 0,C 180,E1 -21298.478,E2 -21298.478} C_VEL
LIN {X 0,Y 213.172,Z 439.932,A -85,B 0,C 180,E1 -21299.175,E2 -21299.175} C_VEL
LIN {X 0,Y 209.613,Z 447.951,A -85,B 0,C 180,E1 -21302.004,E2 -21302.004} C_VEL
LIN {X 0,Y 205.927,Z 455.617,A -85,B 0,C 180,E1 -21305.286,E2 -21305.286} C_VEL
LIN {X 0,Y 202.923,Z 461.972,A -85,B 0,C 180,E1 -21308.675,E2 -21308.675} C_VEL
LIN {X 0,Y 200.42,Z 467.816,A -85,B 0,C 180,E1 -21312.658,E2 -21312.658} C_VEL
LIN {X 0,Y 198.99,Z 471.291,A -85,B 0,C 180,E1 -21315.686,E2 -21315.686} C_VEL
LIN {X 0,Y 197.834,Z 474.801,A -85,B 0,C 180,E1 -21319.768,E2 -21319.768} C_VEL
LIN {X 0,Y 197.268,Z 477.11,A -85,B 0,C 180,E1 -21323.864,E2 -21323.864} C_VEL
LIN {X 0,Y 197.171,Z 478.27,A -85,B 0,C 180,E1 -21327.957,E2 -21327.957} C_VEL
LIN {X 0,Y 197.24,Z 478.422,A -85,B 0,C 180,E1 -21329.999,E2 -21329.999} C_VEL
LIN {X 0,Y 197.171,Z 477.817,A -85,B 0,C 180,E1 -21334.087,E2 -21334.087} C_VEL
LIN {X 0,Y 197.472,Z 476.069,A -85,B 0,C 180,E1 -21338.183,E2 -21338.183} C_VEL
LIN {X 0,Y 198.312,Z 473.154,A -85,B 0,C 180,E1 -21342.276,E2 -21342.276} C_VEL
LIN {X 0,Y 199.942,Z 469.005,A -85,B 0,C 180,E1 -21346.331,E2 -21346.331} C_VEL
LIN {X 0,Y 202.245,Z 463.509,A -85,B 0,C 180,E1 -21350.333,E2 -21350.333} C_VEL
LIN {X 0,Y 205.444,Z 456.518,A -85,B 0,C 180,E1 -21354.235,E2 -21354.235} C_VEL
LIN {X 0,Y 208.996,Z 449.041,A -85,B 0,C 180,E1 -21357.539,E2 -21357.539} C_VEL
LIN {X 0,Y 212.97,Z 440.391,A -85,B 0,C 180,E1 -21360.614,E2 -21360.614} C_VEL
LIN {X 0,Y 217.139,Z 430.822,A -85,B 0,C 180,E1 -21363.381,E2 -21363.381} C_VEL
LIN {X 0,Y 221.631,Z 419.978,A -85,B 0,C 180,E1 -21365.918,E2 -21365.918} C_VEL
LIN {X 0,Y 226.168,Z 408.14,A -85,B 0,C 180,E1 -21368.139,E2 -21368.139} C_VEL
LIN {X 0,Y 227.22,Z 404.866,A -85,B 0,C 180,E1 -21368.712,E2 -21368.712} C_VEL
LIN {X 0,Y 227.089,Z 395.142,A -85,B 0,C 180,E1 -21370.826,E2 -21370.826} C_VEL
LIN {X 0,Y 226.008,Z 383.258,A -85,B 0,C 180,E1 -21373.344,E2 -21373.344} C_VEL
LIN {X 0,Y 223.711,Z 370.942,A -85,B 0,C 180,E1 -21375.968,E2 -21375.968} C_VEL
LIN {X 0,Y 220.991,Z 361.327,A -85,B 0,C 180,E1 -21378.099,E2 -21378.099} C_VEL
LIN {X 0,Y 217.658,Z 353.286,A -85,B 0,C 180,E1 -21380.135,E2 -21380.135} C_VEL
LIN {X 0,Y 213.627,Z 345.216,A -85,B 0,C 180,E1 -21382.392,E2 -21382.392} C_VEL
LIN {X 0,Y 210.438,Z 339.711,A -85,B 0,C 180,E1 -21384.126,E2 -21384.126} C_VEL
LIN {X 0,Y 207.996,Z 335.455,A -85,B 0,C 180,E1 -21385.457,E2 -21385.457} C_VEL
LIN {X 0,Y 205.243,Z 331.737,A -85,B 0,C 180,E1 -21386.937,E2 -21386.937} C_VEL
LIN {X 0,Y 204.068,Z 329.387,A -85,B 0,C 180,E1 -21387.625,E2 -21387.625} C_VEL
LIN {X 0,Y 201.459,Z 326.608,A -85,B 0,C 180,E1 -21389.032,E2 -21389.032} C_VEL
LIN {X 0,Y 200.133,Z 323.306,A -85,B 0,C 180,E1 -21389.973,E2 -21389.973} C_VEL
LIN {X 0,Y 199.868,Z 321.293,A -85,B 0,C 180,E1 -21395.042,E2 -21395.042} C_VEL
LIN {X 0,Y 199.751,Z 320.533,A -85,B 0,C 180,E1 -21397.231,E2 -21397.231} C_VEL
LIN {X 0,Y 199.792,Z 320.223,A -85,B 0,C 180,E1 -21401.757,E2 -21401.757} C_VEL
LIN {X 0,Y 199.828,Z 320.215,A -85,B 0,C 180,E1 -21405.748,E2 -21405.748} C_VEL
LIN {X 0,Y 200.018,Z 320.195,A -85,B 0,C 180,E1 -21409.882,E2 -21409.882} C_VEL
LIN {X 0,Y 200.005,Z 320.191,A -85,B 0,C 180,E1 -21413.949,E2 -21413.949} C_VEL
LIN {X 0,Y 200.314,Z 320.151,A -85,B 0,C 180,E1 -21417.99,E2 -21417.99} C_VEL
LIN {X 0,Y 200.467,Z 320.139,A -85,B 0,C 180,E1 -21420,E2 -21420} C_VEL
LIN {X 0,Y 200.015,Z 320.194,A -85,B 0,C 180,E1 -21424.03,E2 -21424.03} C_VEL
LIN {X 0,Y 200.068,Z 320.182,A -85,B 0,C 180,E1 -21428.078,E2 -21428.078} C_VEL
LIN {X 0,Y 199.868,Z 320.208,A -85,B 0,C 180,E1 -21432.18,E2 -21432.18} C_VEL
LIN {X 0,Y 199.799,Z 320.223,A -85,B 0,C 180,E1 -21436.344,E2 -21436.344} C_VEL
LIN {X 0,Y 199.82,Z 320.217,A -85,B 0,C 180,E1 -21438.454,E2 -21438.454} C_VEL
LIN {X 0,Y 199.733,Z 320.231,A -85,B 0,C 180,E1 -21443.818,E2 -21443.818} C_VEL
LIN {X 0,Y 199.725,Z 320.531,A -85,B 0,C 180,E1 -21447.223,E2 -21447.223} C_VEL
LIN {X 0,Y 199.862,Z 321.56,A -85,B 0,C 180,E1 -21450,E2 -21450} C_VEL
LIN {X 0,Y 200.972,Z 324.343,A -85,B 0,C 180,E1 -21450.76,E2 -21450.76} C_VEL
LIN {X 0,Y 203.547,Z 327.177,A -85,B 0,C 180,E1 -21452.182,E2 -21452.182} C_VEL
LIN {X 0,Y 204.175,Z 327.937,A -85,B 0,C 180,E1 -21452.52,E2 -21452.52} C_VEL
LIN {X 0,Y 206.217,Z 331.521,A -85,B 0,C 180,E1 -21453.702,E2 -21453.702} C_VEL
LIN {X 0,Y 207.865,Z 333.517,A -85,B 0,C 180,E1 -21454.568,E2 -21454.568} C_VEL
LIN {X 0,Y 210.157,Z 337.381,A -85,B 0,C 180,E1 -21455.819,E2 -21455.819} C_VEL
LIN {X 0,Y 211.248,Z 339.137,A -85,B 0,C 180,E1 -21456.416,E2 -21456.416} C_VEL
LIN {X 0,Y 214.723,Z 345.274,A -85,B 0,C 180,E1 -21458.306,E2 -21458.306} C_VEL
LIN {X 0,Y 218.497,Z 352.75,A -85,B 0,C 180,E1 -21460.433,E2 -21460.433} C_VEL
LIN {X 0,Y 222.249,Z 362.218,A -85,B 0,C 180,E1 -21462.836,E2 -21462.836} C_VEL
LIN {X 0,Y 224.964,Z 372.209,A -85,B 0,C 180,E1 -21465.1,E2 -21465.1} C_VEL
LIN {X 0,Y 227.061,Z 383.829,A -85,B 0,C 180,E1 -21467.645,E2 -21467.645} C_VEL
LIN {X 0,Y 228.137,Z 394.713,A -85,B 0,C 180,E1 -21470.043,E2 -21470.043} C_VEL
LIN {X 0,Y 228.249,Z 399.445,A -85,B 0,C 180,E1 -21471.108,E2 -21471.108} C_VEL
LIN {X 0,Y 225.844,Z 406.831,A -85,B 0,C 180,E1 -21472.361,E2 -21472.361} C_VEL
LIN {X 0,Y 221.491,Z 418.27,A -85,B 0,C 180,E1 -21474.616,E2 -21474.616} C_VEL
LIN {X 0,Y 217.111,Z 428.775,A -85,B 0,C 180,E1 -21477.166,E2 -21477.166} C_VEL
LIN {X 0,Y 212.554,Z 439.044,A -85,B 0,C 180,E1 -21480.268,E2 -21480.268} C_VEL
LIN {X 0,Y 208.488,Z 447.568,A -85,B 0,C 180,E1 -21483.472,E2 -21483.472} C_VEL
LIN {X 0,Y 205.127,Z 454.66,A -85,B 0,C 180,E1 -21486.797,E2 -21486.797} C_VEL
LIN {X 0,Y 202.064,Z 461.24,A -85,B 0,C 180,E1 -21490.707,E2 -21490.707} C_VEL
LIN {X 0,Y 199.797,Z 466.382,A -85,B 0,C 180,E1 -21494.704,E2 -21494.704} C_VEL
LIN {X 0,Y 198.616,Z 469.344,A -85,B 0,C 180,E1 -21497.743,E2 -21497.743} C_VEL
LIN {X 0,Y 197.649,Z 472.242,A -85,B 0,C 180,E1 -21501.824,E2 -21501.824} C_VEL
LIN {X 0,Y 197.242,Z 474.024,A -85,B 0,C 180,E1 -21506.098,E2 -21506.098} C_VEL
LIN {X 0,Y 197.248,Z 474.586,A -85,B 0,C 180,E1 -21510.001,E2 -21510.001} C_VEL
LIN {X 0,Y 197.247,Z 474.016,A -85,B 0,C 180,E1 -21514.087,E2 -21514.087} C_VEL
LIN {X 0,Y 197.635,Z 472.324,A -85,B 0,C 180,E1 -21518.178,E2 -21518.178} C_VEL
LIN {X 0,Y 198.583,Z 469.469,A -85,B 0,C 180,E1 -21522.26,E2 -21522.26} C_VEL
LIN {X 0,Y 200.284,Z 465.382,A -85,B 0,C 180,E1 -21526.304,E2 -21526.304} C_VEL
LIN {X 0,Y 202.688,Z 459.965,A -85,B 0,C 180,E1 -21530.289,E2 -21530.289} C_VEL
LIN {X 0,Y 205.936,Z 453.063,A -85,B 0,C 180,E1 -21534.175,E2 -21534.175} C_VEL
LIN {X 0,Y 210,Z 444.45,A -85,B 0,C 180,E1 -21537.939,E2 -21537.939} C_VEL
LIN {X 0,Y 214.348,Z 435.291,A -85,B 0,C 180,E1 -21541.092,E2 -21541.092} C_VEL
LIN {X 0,Y 218.374,Z 425.967,A -85,B 0,C 180,E1 -21543.722,E2 -21543.722} C_VEL
LIN {X 0,Y 223.277,Z 413.897,A -85,B 0,C 180,E1 -21546.45,E2 -21546.45} C_VEL
LIN {X 0,Y 227.915,Z 401.381,A -85,B 0,C 180,E1 -21548.683,E2 -21548.683} C_VEL
LIN {X 0,Y 228.322,Z 399.989,A -85,B 0,C 180,E1 -21548.907,E2 -21548.907} C_VEL
LIN {X 0,Y 227.817,Z 389.486,A -85,B 0,C 180,E1 -21551.254,E2 -21551.254} C_VEL
LIN {X 0,Y 226.227,Z 378.039,A -85,B 0,C 180,E1 -21553.761,E2 -21553.761} C_VEL
LIN {X 0,Y 223.967,Z 367.86,A -85,B 0,C 180,E1 -21556.03,E2 -21556.03} C_VEL
LIN {X 0,Y 221.124,Z 358.897,A -85,B 0,C 180,E1 -21558.13,E2 -21558.13} C_VEL
LIN {X 0,Y 217.351,Z 350.397,A -85,B 0,C 180,E1 -21560.387,E2 -21560.387} C_VEL
LIN {X 0,Y 213.283,Z 342.63,A -85,B 0,C 180,E1 -21562.662,E2 -21562.662} C_VEL
LIN {X 0,Y 210.443,Z 337.714,A -85,B 0,C 180,E1 -21564.237,E2 -21564.237} C_VEL
LIN {X 0,Y 208.119,Z 334.091,A -85,B 0,C 180,E1 -21565.48,E2 -21565.48} C_VEL
LIN {X 0,Y 207.237,Z 332.658,A -85,B 0,C 180,E1 -21565.974,E2 -21565.974} C_VEL
LIN {X 0,Y 204.774,Z 329.23,A -85,B 0,C 180,E1 -21567.335,E2 -21567.335} C_VEL
LIN {X 0,Y 203.865,Z 327.403,A -85,B 0,C 180,E1 -21567.877,E2 -21567.877} C_VEL
LIN {X 0,Y 201.264,Z 324.817,A -85,B 0,C 180,E1 -21569.29,E2 -21569.29} C_VEL
LIN {X 0,Y 200.027,Z 322.295,A -85,B 0,C 180,E1 -21570.1,E2 -21570.1} C_VEL
LIN {X 0,Y 199.802,Z 321.46,A -85,B 0,C 180,E1 -21570.353,E2 -21570.353} C_VEL
LIN {X 0,Y 199.714,Z 320.628,A -85,B 0,C 180,E1 -21572.776,E2 -21572.776} C_VEL
LIN {X 0,Y 199.708,Z 320.232,A -85,B 0,C 180,E1 -21576.202,E2 -21576.202} C_VEL
LIN {X 0,Y 199.797,Z 320.221,A -85,B 0,C 180,E1 -21581.758,E2 -21581.758} C_VEL
LIN {X 0,Y 199.832,Z 320.218,A -85,B 0,C 180,E1 -21585.748,E2 -21585.748} C_VEL
LIN {X 0,Y 200.023,Z 320.193,A -85,B 0,C 180,E1 -21589.882,E2 -21589.882} C_VEL
LIN {X 0,Y 200.01,Z 320.195,A -85,B 0,C 180,E1 -21593.949,E2 -21593.949} C_VEL
LIN {X 0,Y 200.318,Z 320.158,A -85,B 0,C 180,E1 -21597.989,E2 -21597.989} C_VEL
LIN {X 0,Y 200.47,Z 320.139,A -85,B 0,C 180,E1 -21600,E2 -21600} C_VEL
LIN {X 0,Y 200.02,Z 320.196,A -85,B 0,C 180,E1 -21604.029,E2 -21604.029} C_VEL
LIN {X 0,Y 200.077,Z 320.189,A -85,B 0,C 180,E1 -21608.077,E2 -21608.077} C_VEL
LIN {X 0,Y 199.874,Z 320.213,A -85,B 0,C 180,E1 -21612.179,E2 -21612.179} C_VEL
LIN {X 0,Y 199.804,Z 320.223,A -85,B 0,C 180,E1 -21616.343,E2 -21616.343} C_VEL
LIN {X 0,Y 199.691,Z 320.236,A -85,B 0,C 180,E1 -21620.606,E2 -21620.606} C_VEL
LIN {X 0,Y 199.83,Z 320.967,A -85,B 0,C 180,E1 -21623.877,E2 -21623.877} C_VEL
LIN {X 0,Y 200.045,Z 322.745,A -85,B 0,C 180,E1 -21628.562,E2 -21628.562} C_VEL
LIN {X 0,Y 200.148,Z 323.491,A -85,B 0,C 180,E1 -21629.952,E2 -21629.952} C_VEL
LIN {X 0,Y 201.263,Z 326.267,A -85,B 0,C 180,E1 -21630.71,E2 -21630.71} C_VEL
LIN {X 0,Y 203.636,Z 329.043,A -85,B 0,C 180,E1 -21632.029,E2 -21632.029} C_VEL
LIN {X 0,Y 204.385,Z 329.889,A -85,B 0,C 180,E1 -21632.427,E2 -21632.427} C_VEL
LIN {X 0,Y 206.398,Z 333.552,A -85,B 0,C 180,E1 -21633.595,E2 -21633.595} C_VEL
LIN {X 0,Y 208.143,Z 335.75,A -85,B 0,C 180,E1 -21634.515,E2 -21634.515} C_VEL
LIN {X 0,Y 210.538,Z 339.845,A -85,B 0,C 180,E1 -21635.818,E2 -21635.818} C_VEL
LIN {X 0,Y 211.891,Z 342.304,A -85,B 0,C 180,E1 -21636.582,E2 -21636.582} C_VEL
LIN {X 0,Y 214.388,Z 346.686,A -85,B 0,C 180,E1 -21637.927,E2 -21637.927} C_VEL
LIN {X 0,Y 218.269,Z 354.309,A -85,B 0,C 180,E1 -21640.089,E2 -21640.089} C_VEL
LIN {X 0,Y 222.08,Z 364.489,A -85,B 0,C 180,E1 -21642.567,E2 -21642.567} C_VEL
LIN {X 0,Y 224.573,Z 374.545,A -85,B 0,C 180,E1 -21644.76,E2 -21644.76} C_VEL
LIN {X 0,Y 226.444,Z 385.709,A -85,B 0,C 180,E1 -21647.126,E2 -21647.126} C_VEL
LIN {X 0,Y 227.338,Z 398.218,A -85,B 0,C 180,E1 -21649.79,E2 -21649.79} C_VEL
LIN {X 0,Y 227.347,Z 404.936,A -85,B 0,C 180,E1 -21651.27,E2 -21651.27} C_VEL
LIN {X 0,Y 222.874,Z 417.216,A -85,B 0,C 180,E1 -21653.473,E2 -21653.473} C_VEL
LIN {X 0,Y 217.87,Z 429.361,A -85,B 0,C 180,E1 -21656.189,E2 -21656.189} C_VEL
LIN {X 0,Y 213.172,Z 439.932,A -85,B 0,C 180,E1 -21659.175,E2 -21659.175} C_VEL
LIN {X 0,Y 211.02,Z 443.563,A -85,B 0,C 180,E1 -21660.308,E2 -21660.308} C_VEL
LIN {X 0,Y 205.852,Z 449.21,A -85,B 0,C 180,E1 -21662.041,E2 -21662.041} C_VEL
LIN {X 0,Y 200.69,Z 454.38,A -85,B 0,C 180,E1 -21663.927,E2 -21663.927} C_VEL
LIN {X 0,Y 198.597,Z 457.244,A -85,B 0,C 180,E1 -21665.281,E2 -21665.281} C_VEL
LIN {X 0,Y 195.095,Z 464.357,A -85,B 0,C 180,E1 -21669.489,E2 -21669.489} C_VEL
LIN {X 0,Y 192.59,Z 470.153,A -85,B 0,C 180,E1 -21674.115,E2 -21674.115} C_VEL
LIN {X 0,Y 191.32,Z 473.132,A -85,B 0,C 180,E1 -21677.267,E2 -21677.267} C_VEL
LIN {X 0,Y 190.433,Z 476.033,A -85,B 0,C 180,E1 -21681.51,E2 -21681.51} C_VEL
LIN {X 0,Y 190.084,Z 477.762,A -85,B 0,C 180,E1 -21685.759,E2 -21685.759} C_VEL
LIN {X 0,Y 190.148,Z 478.353,A -85,B 0,C 180,E1 -21689.999,E2 -21689.999} C_VEL
LIN {X 0,Y 190.084,Z 477.748,A -85,B 0,C 180,E1 -21694.24,E2 -21694.24} C_VEL
LIN {X 0,Y 190.432,Z 476,A -85,B 0,C 180,E1 -21698.488,E2 -21698.488} C_VEL
LIN {X 0,Y 191.319,Z 473.084,A -85,B 0,C 180,E1 -21702.732,E2 -21702.732} C_VEL
LIN {X 0,Y 193.088,Z 468.935,A -85,B 0,C 180,E1 -21706.928,E2 -21706.928} C_VEL
LIN {X 0,Y 195.538,Z 463.438,A -85,B 0,C 180,E1 -21711.063,E2 -21711.063} C_VEL
LIN {X 0,Y 198.947,Z 456.447,A -85,B 0,C 180,E1 -21715.081,E2 -21715.081} C_VEL
LIN {X 0,Y 202.704,Z 448.97,A -85,B 0,C 180,E1 -21718.471,E2 -21718.471} C_VEL
LIN {X 0,Y 207.133,Z 439.712,A -85,B 0,C 180,E1 -21721.83,E2 -21721.83} C_VEL
LIN {X 0,Y 211.979,Z 429.115,A -85,B 0,C 180,E1 -21724.882,E2 -21724.882} C_VEL
LIN {X 0,Y 216.762,Z 417.953,A -85,B 0,C 180,E1 -21727.438,E2 -21727.438} C_VEL
LIN {X 0,Y 221.07,Z 406.893,A -85,B 0,C 180,E1 -21729.479,E2 -21729.479} C_VEL
LIN {X 0,Y 221.136,Z 396.495,A -85,B 0,C 180,E1 -21731.865,E2 -21731.865} C_VEL
LIN {X 0,Y 220.389,Z 386.256,A -85,B 0,C 180,E1 -21734.153,E2 -21734.153} C_VEL
LIN {X 0,Y 218.752,Z 375.81,A -85,B 0,C 180,E1 -21736.493,E2 -21736.493} C_VEL
LIN {X 0,Y 216.403,Z 366.302,A -85,B 0,C 180,E1 -21738.716,E2 -21738.716} C_VEL
LIN {X 0,Y 213.619,Z 358.728,A -85,B 0,C 180,E1 -21740.705,E2 -21740.705} C_VEL
LIN {X 0,Y 209.225,Z 349.669,A -85,B 0,C 180,E1 -21743.441,E2 -21743.441} C_VEL
LIN {X 0,Y 206.775,Z 345.113,A -85,B 0,C 180,E1 -21744.927,E2 -21744.927} C_VEL
LIN {X 0,Y 204.205,Z 340.532,A -85,B 0,C 180,E1 -21746.514,E2 -21746.514} C_VEL
LIN {X 0,Y 201.747,Z 336.708,A -85,B 0,C 180,E1 -21747.984,E2 -21747.984} C_VEL
LIN {X 0,Y 200.947,Z 335.213,A -85,B 0,C 180,E1 -21748.505,E2 -21748.505} C_VEL
LIN {X 0,Y 198.523,Z 332.128,A -85,B 0,C 180,E1 -21749.997,E2 -21749.997} C_VEL
LIN {X 0,Y 197.241,Z 329.459,A -85,B 0,C 180,E1 -21750.881,E2 -21750.881} C_VEL
LIN {X 0,Y 194.634,Z 326.957,A -85,B 0,C 180,E1 -21752.515,E2 -21752.515} C_VEL
LIN {X 0,Y 193.126,Z 323.903,A -85,B 0,C 180,E1 -21753.672,E2 -21753.672} C_VEL
LIN {X 0,Y 192.945,Z 323.146,A -85,B 0,C 180,E1 -21753.936,E2 -21753.936} C_VEL
LIN {X 0,Y 192.868,Z 322.29,A -85,B 0,C 180,E1 -21756.37,E2 -21756.37} C_VEL
LIN {X 0,Y 192.689,Z 321.106,A -85,B 0,C 180,E1 -21760.837,E2 -21760.837} C_VEL
LIN {X 0,Y 192.757,Z 321.095,A -85,B 0,C 180,E1 -21765.213,E2 -21765.213} C_VEL
LIN {X 0,Y 192.94,Z 321.078,A -85,B 0,C 180,E1 -21769.567,E2 -21769.567} C_VEL
LIN {X 0,Y 192.968,Z 321.068,A -85,B 0,C 180,E1 -21773.727,E2 -21773.727} C_VEL
LIN {X 0,Y 193.255,Z 321.03,A -85,B 0,C 180,E1 -21777.916,E2 -21777.916} C_VEL
LIN {X 0,Y 193.432,Z 321.015,A -85,B 0,C 180,E1 -21780,E2 -21780} C_VEL
LIN {X 0,Y 192.96,Z 321.073,A -85,B 0,C 180,E1 -21784.178,E2 -21784.178} C_VEL
LIN {X 0,Y 193.019,Z 321.06,A -85,B 0,C 180,E1 -21788.375,E2 -21788.375} C_VEL
LIN {X 0,Y 192.795,Z 321.092,A -85,B 0,C 180,E1 -21792.634,E2 -21792.634} C_VEL
LIN {X 0,Y 192.765,Z 321.096,A -85,B 0,C 180,E1 -21796.958,E2 -21796.958} C_VEL
LIN {X 0,Y 192.638,Z 321.114,A -85,B 0,C 180,E1 -21801.397,E2 -21801.397} C_VEL
LIN {X 0,Y 192.66,Z 321.111,A -85,B 0,C 180,E1 -21804.225,E2 -21804.225} C_VEL
LIN {X 0,Y 192.725,Z 321.828,A -85,B 0,C 180,E1 -21806.096,E2 -21806.096} C_VEL
LIN {X 0,Y 193.694,Z 324.264,A -85,B 0,C 180,E1 -21806.899,E2 -21806.899} C_VEL
LIN {X 0,Y 196.229,Z 327.169,A -85,B 0,C 180,E1 -21808.59,E2 -21808.59} C_VEL
LIN {X 0,Y 197.201,Z 327.987,A -85,B 0,C 180,E1 -21809.177,E2 -21809.177} C_VEL
LIN {X 0,Y 199.031,Z 331.401,A -85,B 0,C 180,E1 -21810.431,E2 -21810.431} C_VEL
LIN {X 0,Y 201.241,Z 334.006,A -85,B 0,C 180,E1 -21811.764,E2 -21811.764} C_VEL
LIN {X 0,Y 203.604,Z 337.964,A -85,B 0,C 180,E1 -21813.228,E2 -21813.228} C_VEL
LIN {X 0,Y 204.772,Z 339.694,A -85,B 0,C 180,E1 -21813.935,E2 -21813.935} C_VEL
LIN {X 0,Y 207.773,Z 344.921,A -85,B 0,C 180,E1 -21815.751,E2 -21815.751} C_VEL
LIN {X 0,Y 211.427,Z 351.836,A -85,B 0,C 180,E1 -21817.994,E2 -21817.994} C_VEL
LIN {X 0,Y 215.557,Z 361.184,A -85,B 0,C 180,E1 -21820.699,E2 -21820.699} C_VEL
LIN {X 0,Y 218.292,Z 369.884,A -85,B 0,C 180,E1 -21822.912,E2 -21822.912} C_VEL
LIN {X 0,Y 220.361,Z 379.612,A -85,B 0,C 180,E1 -21825.204,E2 -21825.204} C_VEL
LIN {X 0,Y 221.805,Z 390.79,A -85,B 0,C 180,E1 -21827.798,E2 -21827.798} C_VEL
LIN {X 0,Y 222.201,Z 400.904,A -85,B 0,C 180,E1 -21830.156,E2 -21830.156} C_VEL
LIN {X 0,Y 221.533,Z 403.39,A -85,B 0,C 180,E1 -21830.62,E2 -21830.62} C_VEL
LIN {X 0,Y 217.281,Z 414.448,A -85,B 0,C 180,E1 -21832.667,E2 -21832.667} C_VEL
LIN {X 0,Y 212.581,Z 425.594,A -85,B 0,C 180,E1 -21835.231,E2 -21835.231} C_VEL
LIN {X 0,Y 207.708,Z 436.416,A -85,B 0,C 180,E1 -21838.37,E2 -21838.37} C_VEL
LIN {X 0,Y 203.227,Z 445.407,A -85,B 0,C 180,E1 -21841.609,E2 -21841.609} C_VEL
LIN {X 0,Y 199.513,Z 452.856,A -85,B 0,C 180,E1 -21844.996,E2 -21844.996} C_VEL
LIN {X 0,Y 196.057,Z 459.818,A -85,B 0,C 180,E1 -21848.995,E2 -21848.995} C_VEL
LIN {X 0,Y 193.479,Z 465.287,A -85,B 0,C 180,E1 -21853.108,E2 -21853.108} C_VEL
LIN {X 0,Y 191.643,Z 469.415,A -85,B 0,C 180,E1 -21857.29,E2 -21857.29} C_VEL
LIN {X 0,Y 190.605,Z 472.312,A -85,B 0,C 180,E1 -21861.52,E2 -21861.52} C_VEL
LIN {X 0,Y 190.166,Z 474.051,A -85,B 0,C 180,E1 -21865.762,E2 -21865.762} C_VEL
LIN {X 0,Y 190.157,Z 474.655,A -85,B 0,C 180,E1 -21870.001,E2 -21870.001} C_VEL
LIN {X 0,Y 190.164,Z 474.085,A -85,B 0,C 180,E1 -21874.24,E2 -21874.24} C_VEL
LIN {X 0,Y 190.593,Z 472.393,A -85,B 0,C 180,E1 -21878.483,E2 -21878.483} C_VEL
LIN {X 0,Y 191.615,Z 469.537,A -85,B 0,C 180,E1 -21882.714,E2 -21882.714} C_VEL
LIN {X 0,Y 193.429,Z 465.45,A -85,B 0,C 180,E1 -21886.899,E2 -21886.899} C_VEL
LIN {X 0,Y 195.964,Z 460.033,A -85,B 0,C 180,E1 -21891.017,E2 -21891.017} C_VEL
LIN {X 0,Y 199.453,Z 453.131,A -85,B 0,C 180,E1 -21895.014,E2 -21895.014} C_VEL
LIN {X 0,Y 203.712,Z 444.517,A -85,B 0,C 180,E1 -21898.882,E2 -21898.882} C_VEL
LIN {X 0,Y 207.611,Z 436.773,A -85,B 0,C 180,E1 -21901.648,E2 -21901.648} C_VEL
LIN {X 0,Y 211.732,Z 427.658,A -85,B 0,C 180,E1 -21904.353,E2 -21904.353} C_VEL
LIN {X 0,Y 216.386,Z 416.905,A -85,B 0,C 180,E1 -21906.932,E2 -21906.932} C_VEL
LIN {X 0,Y 220.984,Z 405.167,A -85,B 0,C 180,E1 -21909.205,E2 -21909.205} C_VEL
LIN {X 0,Y 222.271,Z 401.454,A -85,B 0,C 180,E1 -21909.856,E2 -21909.856} C_VEL
LIN {X 0,Y 221.864,Z 390.51,A -85,B 0,C 180,E1 -21912.41,E2 -21912.41} C_VEL
LIN {X 0,Y 220.334,Z 378.847,A -85,B 0,C 180,E1 -21915.112,E2 -21915.112} C_VEL
LIN {X 0,Y 217.869,Z 367.995,A -85,B 0,C 180,E1 -21917.709,E2 -21917.709} C_VEL
LIN {X 0,Y 215.126,Z 359.877,A -85,B 0,C 180,E1 -21919.818,E2 -21919.818} C_VEL
LIN {X 0,Y 210.854,Z 350.693,A -85,B 0,C 180,E1 -21922.544,E2 -21922.544} C_VEL
LIN {X 0,Y 208.877,Z 347.031,A -85,B 0,C 180,E1 -21923.75,E2 -21923.75} C_VEL
LIN {X 0,Y 206.545,Z 342.778,A -85,B 0,C 180,E1 -21925.179,E2 -21925.179} C_VEL
LIN {X 0,Y 203.798,Z 338.133,A -85,B 0,C 180,E1 -21926.881,E2 -21926.881} C_VEL
LIN {X 0,Y 201.3,Z 334.121,A -85,B 0,C 180,E1 -21928.419,E2 -21928.419} C_VEL
LIN {X 0,Y 200.36,Z 332.918,A -85,B 0,C 180,E1 -21928.99,E2 -21928.99} C_VEL
LIN {X 0,Y 198.101,Z 329.941,A -85,B 0,C 180,E1 -21930.426,E2 -21930.426} C_VEL
LIN {X 0,Y 197.067,Z 327.775,A -85,B 0,C 180,E1 -21931.154,E2 -21931.154} C_VEL
LIN {X 0,Y 194.322,Z 325.223,A -85,B 0,C 180,E1 -21932.904,E2 -21932.904} C_VEL
LIN {X 0,Y 192.969,Z 322.808,A -85,B 0,C 180,E1 -21933.939,E2 -21933.939} C_VEL
LIN {X 0,Y 192.658,Z 321.616,A -85,B 0,C 180,E1 -21934.288,E2 -21934.288} C_VEL
LIN {X 0,Y 192.679,Z 321.109,A -85,B 0,C 180,E1 -21936.345,E2 -21936.345} C_VEL
LIN {X 0,Y 192.733,Z 321.099,A -85,B 0,C 180,E1 -21941.458,E2 -21941.458} C_VEL
LIN {X 0,Y 192.761,Z 321.1,A -85,B 0,C 180,E1 -21945.213,E2 -21945.213} C_VEL
LIN {X 0,Y 192.946,Z 321.075,A -85,B 0,C 180,E1 -21949.567,E2 -21949.567} C_VEL
LIN {X 0,Y 192.973,Z 321.072,A -85,B 0,C 180,E1 -21953.727,E2 -21953.727} C_VEL
LIN {X 0,Y 193.26,Z 321.036,A -85,B 0,C 180,E1 -21957.916,E2 -21957.916} C_VEL
LIN {X 0,Y 193.435,Z 321.015,A -85,B 0,C 180,E1 -21960,E2 -21960} C_VEL
LIN {X 0,Y 192.965,Z 321.075,A -85,B 0,C 180,E1 -21964.177,E2 -21964.177} C_VEL
LIN {X 0,Y 193.027,Z 321.066,A -85,B 0,C 180,E1 -21968.374,E2 -21968.374} C_VEL
LIN {X 0,Y 192.802,Z 321.094,A -85,B 0,C 180,E1 -21972.633,E2 -21972.633} C_VEL
LIN {X 0,Y 192.757,Z 321.101,A -85,B 0,C 180,E1 -21976.958,E2 -21976.958} C_VEL
LIN {X 0,Y 192.691,Z 321.108,A -85,B 0,C 180,E1 -21979.163,E2 -21979.163} C_VEL
LIN {X 0,Y 192.894,Z 322.605,A -85,B 0,C 180,E1 -21984.375,E2 -21984.375} C_VEL
LIN {X 0,Y 192.951,Z 323.217,A -85,B 0,C 180,E1 -21985.99,E2 -21985.99} C_VEL
LIN {X 0,Y 193.914,Z 325.763,A -85,B 0,C 180,E1 -21986.793,E2 -21986.793} C_VEL
LIN {X 0,Y 196.039,Z 328.525,A -85,B 0,C 180,E1 -21988.244,E2 -21988.244} C_VEL
LIN {X 0,Y 197.427,Z 329.753,A -85,B 0,C 180,E1 -21989.09,E2 -21989.09} C_VEL
LIN {X 0,Y 199.402,Z 333.492,A -85,B 0,C 180,E1 -21990.441,E2 -21990.441} C_VEL
LIN {X 0,Y 201.402,Z 335.822,A -85,B 0,C 180,E1 -21991.636,E2 -21991.636} C_VEL
LIN {X 0,Y 203.492,Z 339.592,A -85,B 0,C 180,E1 -21992.953,E2 -21992.953} C_VEL
LIN {X 0,Y 204.911,Z 341.649,A -85,B 0,C 180,E1 -21993.798,E2 -21993.798} C_VEL
LIN {X 0,Y 208.115,Z 347.496,A -85,B 0,C 180,E1 -21995.754,E2 -21995.754} C_VEL
LIN {X 0,Y 211.005,Z 353.116,A -85,B 0,C 180,E1 -21997.545,E2 -21997.545} C_VEL
LIN {X 0,Y 214.426,Z 360.582,A -85,B 0,C 180,E1 -21999.727,E2 -21999.727} C_VEL
LIN {X 0,Y 217.348,Z 369.373,A -85,B 0,C 180,E1 -22001.951,E2 -22001.951} C_VEL
LIN {X 0,Y 219.222,Z 377.67,A -85,B 0,C 180,E1 -22003.867,E2 -22003.867} C_VEL
LIN {X 0,Y 220.789,Z 388.9,A -85,B 0,C 180,E1 -22006.398,E2 -22006.398} C_VEL
LIN {X 0,Y 221.365,Z 400.462,A -85,B 0,C 180,E1 -22009.001,E2 -22009.001} C_VEL
LIN {X 0,Y 221.1,Z 407.139,A -85,B 0,C 180,E1 -22010.526,E2 -22010.526} C_VEL
LIN {X 0,Y 216.769,Z 418.158,A -85,B 0,C 180,E1 -22012.562,E2 -22012.562} C_VEL
LIN {X 0,Y 211.985,Z 429.294,A -85,B 0,C 180,E1 -22015.117,E2 -22015.117} C_VEL
LIN {X 0,Y 207.406,Z 439.069,A -85,B 0,C 180,E1 -22017.9,E2 -22017.9} C_VEL
LIN {X 0,Y 203.321,Z 447.883,A -85,B 0,C 180,E1 -22021.058,E2 -22021.058} C_VEL
LIN {X 0,Y 199.428,Z 455.548,A -85,B 0,C 180,E1 -22024.424,E2 -22024.424} C_VEL
LIN {X 0,Y 198.597,Z 457.244,A -85,B 0,C 180,E1 -22025.281,E2 -22025.281} C_VEL
LIN {X 0,Y 196.602,Z 459.992,A -85,B 0,C 180,E1 -22026.694,E2 -22026.694} C_VEL
LIN {X 0,Y 191.875,Z 464.114,A -85,B 0,C 180,E1 -22028.965,E2 -22028.965} C_VEL
LIN {X 0,Y 187.427,Z 467.699,A -85,B 0,C 180,E1 -22031.408,E2 -22031.408} C_VEL
LIN {X 0,Y 185.913,Z 469.599,A -85,B 0,C 180,E1 -22033.056,E2 -22033.056} C_VEL
LIN {X 0,Y 184.343,Z 473.063,A -85,B 0,C 180,E1 -22036.776,E2 -22036.776} C_VEL
LIN {X 0,Y 183.382,Z 475.964,A -85,B 0,C 180,E1 -22041.181,E2 -22041.181} C_VEL
LIN {X 0,Y 183.013,Z 477.693,A -85,B 0,C 180,E1 -22045.594,E2 -22045.594} C_VEL
LIN {X 0,Y 183.058,Z 478.284,A -85,B 0,C 180,E1 -22049.999,E2 -22049.999} C_VEL
LIN {X 0,Y 183.012,Z 477.679,A -85,B 0,C 180,E1 -22054.404,E2 -22054.404} C_VEL
LIN {X 0,Y 183.381,Z 475.93,A -85,B 0,C 180,E1 -22058.817,E2 -22058.817} C_VEL
LIN {X 0,Y 184.341,Z 473.014,A -85,B 0,C 180,E1 -22063.222,E2 -22063.222} C_VEL
LIN {X 0,Y 186.223,Z 468.864,A -85,B 0,C 180,E1 -22067.572,E2 -22067.572} C_VEL
LIN {X 0,Y 188.858,Z 463.367,A -85,B 0,C 180,E1 -22071.846,E2 -22071.846} C_VEL
LIN {X 0,Y 192.474,Z 456.376,A -85,B 0,C 180,E1 -22075.986,E2 -22075.986} C_VEL
LIN {X 0,Y 196.461,Z 448.899,A -85,B 0,C 180,E1 -22079.463,E2 -22079.463} C_VEL
LIN {X 0,Y 200.808,Z 440.194,A -85,B 0,C 180,E1 -22082.714,E2 -22082.714} C_VEL
LIN {X 0,Y 205.374,Z 430.678,A -85,B 0,C 180,E1 -22085.572,E2 -22085.572} C_VEL
LIN {X 0,Y 210.26,Z 419.833,A -85,B 0,C 180,E1 -22088.195,E2 -22088.195} C_VEL
LIN {X 0,Y 215.073,Z 407.994,A -85,B 0,C 180,E1 -22090.499,E2 -22090.499} C_VEL
LIN {X 0,Y 215.244,Z 397.397,A -85,B 0,C 180,E1 -22093.067,E2 -22093.067} C_VEL
LIN {X 0,Y 214.639,Z 388.113,A -85,B 0,C 180,E1 -22095.254,E2 -22095.254} C_VEL
LIN {X 0,Y 213.288,Z 378.326,A -85,B 0,C 180,E1 -22097.588,E2 -22097.588} C_VEL
LIN {X 0,Y 211.474,Z 370.216,A -85,B 0,C 180,E1 -22099.607,E2 -22099.607} C_VEL
LIN {X 0,Y 209.094,Z 363.235,A -85,B 0,C 180,E1 -22101.551,E2 -22101.551} C_VEL
LIN {X 0,Y 205.072,Z 354.419,A -85,B 0,C 180,E1 -22104.366,E2 -22104.366} C_VEL
LIN {X 0,Y 202.822,Z 350.062,A -85,B 0,C 180,E1 -22105.881,E2 -22105.881} C_VEL
LIN {X 0,Y 200.695,Z 346.027,A -85,B 0,C 180,E1 -22107.35,E2 -22107.35} C_VEL
LIN {X 0,Y 198.34,Z 341.872,A -85,B 0,C 180,E1 -22108.972,E2 -22108.972} C_VEL
LIN {X 0,Y 195.36,Z 337.427,A -85,B 0,C 180,E1 -22111.018,E2 -22111.018} C_VEL
LIN {X 0,Y 194.318,Z 335.473,A -85,B 0,C 180,E1 -22111.808,E2 -22111.808} C_VEL
LIN {X 0,Y 191.887,Z 332.52,A -85,B 0,C 180,E1 -22113.562,E2 -22113.562} C_VEL
LIN {X 0,Y 190.315,Z 329.463,A -85,B 0,C 180,E1 -22114.858,E2 -22114.858} C_VEL
LIN {X 0,Y 187.216,Z 326.434,A -85,B 0,C 180,E1 -22117.297,E2 -22117.297} C_VEL
LIN {X 0,Y 185.921,Z 323.678,A -85,B 0,C 180,E1 -22118.592,E2 -22118.592} C_VEL
LIN {X 0,Y 185.759,Z 323.002,A -85,B 0,C 180,E1 -22118.863,E2 -22118.863} C_VEL
LIN {X 0,Y 185.701,Z 322.03,A -85,B 0,C 180,E1 -22122.376,E2 -22122.376} C_VEL
LIN {X 0,Y 185.723,Z 321.975,A -85,B 0,C 180,E1 -22126.877,E2 -22126.877} C_VEL
LIN {X 0,Y 185.968,Z 321.939,A -85,B 0,C 180,E1 -22131.306,E2 -22131.306} C_VEL
LIN {X 0,Y 186.199,Z 321.909,A -85,B 0,C 180,E1 -22137.837,E2 -22137.837} C_VEL
LIN {X 0,Y 186.396,Z 321.891,A -85,B 0,C 180,E1 -22140,E2 -22140} C_VEL
LIN {X 0,Y 185.907,Z 321.952,A -85,B 0,C 180,E1 -22144.336,E2 -22144.336} C_VEL
LIN {X 0,Y 185.969,Z 321.938,A -85,B 0,C 180,E1 -22148.695,E2 -22148.695} C_VEL
LIN {X 0,Y 185.723,Z 321.977,A -85,B 0,C 180,E1 -22153.124,E2 -22153.124} C_VEL
LIN {X 0,Y 185.712,Z 321.972,A -85,B 0,C 180,E1 -22157.623,E2 -22157.623} C_VEL
LIN {X 0,Y 185.594,Z 322.005,A -85,B 0,C 180,E1 -22161.157,E2 -22161.157} C_VEL
LIN {X 0,Y 186.276,Z 324.228,A -85,B 0,C 180,E1 -22161.948,E2 -22161.948} C_VEL
LIN {X 0,Y 187.926,Z 326.38,A -85,B 0,C 180,E1 -22163.413,E2 -22163.413} C_VEL
LIN {X 0,Y 190.367,Z 328.362,A -85,B 0,C 180,E1 -22165.269,E2 -22165.269} C_VEL
LIN {X 0,Y 192.176,Z 331.677,A -85,B 0,C 180,E1 -22166.762,E2 -22166.762} C_VEL
LIN {X 0,Y 194.616,Z 334.413,A -85,B 0,C 180,E1 -22168.488,E2 -22168.488} C_VEL
LIN {X 0,Y 196.709,Z 338.025,A -85,B 0,C 180,E1 -22170.013,E2 -22170.013} C_VEL
LIN {X 0,Y 198.284,Z 340.098,A -85,B 0,C 180,E1 -22171.075,E2 -22171.075} C_VEL
LIN {X 0,Y 200.567,Z 344.054,A -85,B 0,C 180,E1 -22172.655,E2 -22172.655} C_VEL
LIN {X 0,Y 204.195,Z 350.655,A -85,B 0,C 180,E1 -22175.13,E2 -22175.13} C_VEL
LIN {X 0,Y 208.328,Z 359.275,A -85,B 0,C 180,E1 -22178.001,E2 -22178.001} C_VEL
LIN {X 0,Y 211.339,Z 366.992,A -85,B 0,C 180,E1 -22180.301,E2 -22180.301} C_VEL
LIN {X 0,Y 213.725,Z 376.126,A -85,B 0,C 180,E1 -22182.705,E2 -22182.705} C_VEL
LIN {X 0,Y 215.356,Z 386.288,A -85,B 0,C 180,E1 -22185.218,E2 -22185.218} C_VEL
LIN {X 0,Y 216.173,Z 396.757,A -85,B 0,C 180,E1 -22187.782,E2 -22187.782} C_VEL
LIN {X 0,Y 216.08,Z 403.463,A -85,B 0,C 180,E1 -22189.422,E2 -22189.422} C_VEL
LIN {X 0,Y 211.668,Z 414.521,A -85,B 0,C 180,E1 -22191.499,E2 -22191.499} C_VEL
LIN {X 0,Y 206.761,Z 425.666,A -85,B 0,C 180,E1 -22194.104,E2 -22194.104} C_VEL
LIN {X 0,Y 201.668,Z 436.488,A -85,B 0,C 180,E1 -22197.307,E2 -22197.307} C_VEL
LIN {X 0,Y 196.956,Z 445.478,A -85,B 0,C 180,E1 -22200.619,E2 -22200.619} C_VEL
LIN {X 0,Y 193.046,Z 452.927,A -85,B 0,C 180,E1 -22204.097,E2 -22204.097} C_VEL
LIN {X 0,Y 189.399,Z 459.889,A -85,B 0,C 180,E1 -22208.22,E2 -22208.22} C_VEL
LIN {X 0,Y 186.649,Z 465.358,A -85,B 0,C 180,E1 -22212.47,E2 -22212.47} C_VEL
LIN {X 0,Y 184.692,Z 469.485,A -85,B 0,C 180,E1 -22216.803,E2 -22216.803} C_VEL
LIN {X 0,Y 183.56,Z 472.381,A -85,B 0,C 180,E1 -22221.192,E2 -22221.192} C_VEL
LIN {X 0,Y 183.08,Z 474.12,A -85,B 0,C 180,E1 -22225.598,E2 -22225.598} C_VEL
LIN {X 0,Y 183.068,Z 474.724,A -85,B 0,C 180,E1 -22230.001,E2 -22230.001} C_VEL
LIN {X 0,Y 183.079,Z 474.154,A -85,B 0,C 180,E1 -22234.404,E2 -22234.404} C_VEL
LIN {X 0,Y 183.55,Z 472.461,A -85,B 0,C 180,E1 -22238.811,E2 -22238.811} C_VEL
LIN {X 0,Y 184.667,Z 469.606,A -85,B 0,C 180,E1 -22243.2,E2 -22243.2} C_VEL
LIN {X 0,Y 186.603,Z 465.519,A -85,B 0,C 180,E1 -22247.536,E2 -22247.536} C_VEL
LIN {X 0,Y 189.368,Z 459.939,A -85,B 0,C 180,E1 -22251.902,E2 -22251.902} C_VEL
LIN {X 0,Y 192.982,Z 453.199,A -85,B 0,C 180,E1 -22255.914,E2 -22255.914} C_VEL
LIN {X 0,Y 197.498,Z 444.584,A -85,B 0,C 180,E1 -22259.881,E2 -22259.881} C_VEL
LIN {X 0,Y 201.539,Z 436.842,A -85,B 0,C 180,E1 -22262.718,E2 -22262.718} C_VEL
LIN {X 0,Y 205.874,Z 427.725,A -85,B 0,C 180,E1 -22265.474,E2 -22265.474} C_VEL
LIN {X 0,Y 210.724,Z 416.971,A -85,B 0,C 180,E1 -22268.098,E2 -22268.098} C_VEL
LIN {X 0,Y 215.533,Z 405.232,A -85,B 0,C 180,E1 -22270.397,E2 -22270.397} C_VEL
LIN {X 0,Y 216.26,Z 402.822,A -85,B 0,C 180,E1 -22270.864,E2 -22270.864} C_VEL
LIN {X 0,Y 215.997,Z 391.827,A -85,B 0,C 180,E1 -22273.565,E2 -22273.565} C_VEL
LIN {X 0,Y 214.732,Z 381.018,A -85,B 0,C 180,E1 -22276.227,E2 -22276.227} C_VEL
LIN {X 0,Y 212.709,Z 371.481,A -85,B 0,C 180,E1 -22278.638,E2 -22278.638} C_VEL
LIN {X 0,Y 210.459,Z 364.302,A -85,B 0,C 180,E1 -22280.618,E2 -22280.618} C_VEL
LIN {X 0,Y 206.381,Z 354.9,A -85,B 0,C 180,E1 -22283.585,E2 -22283.585} C_VEL
LIN {X 0,Y 202.886,Z 348.195,A -85,B 0,C 180,E1 -22285.968,E2 -22285.968} C_VEL
LIN {X 0,Y 200.485,Z 343.865,A -85,B 0,C 180,E1 -22287.624,E2 -22287.624} C_VEL
LIN {X 0,Y 197.7,Z 339.194,A -85,B 0,C 180,E1 -22289.564,E2 -22289.564} C_VEL
LIN {X 0,Y 195.296,Z 335.905,A -85,B 0,C 180,E1 -22291.213,E2 -22291.213} C_VEL
LIN {X 0,Y 194.175,Z 333.805,A -85,B 0,C 180,E1 -22292.078,E2 -22292.078} C_VEL
LIN {X 0,Y 191.521,Z 330.762,A -85,B 0,C 180,E1 -22294.02,E2 -22294.02} C_VEL
LIN {X 0,Y 190.193,Z 328.034,A -85,B 0,C 180,E1 -22295.157,E2 -22295.157} C_VEL
LIN {X 0,Y 187.039,Z 325.483,A -85,B 0,C 180,E1 -22297.638,E2 -22297.638} C_VEL
LIN {X 0,Y 185.873,Z 323.292,A -85,B 0,C 180,E1 -22298.803,E2 -22298.803} C_VEL
LIN {X 0,Y 185.58,Z 321.994,A -85,B 0,C 180,E1 -22299.204,E2 -22299.204} C_VEL
LIN {X 0,Y 185.69,Z 321.98,A -85,B 0,C 180,E1 -22302.375,E2 -22302.375} C_VEL
LIN {X 0,Y 185.727,Z 321.968,A -85,B 0,C 180,E1 -22306.877,E2 -22306.877} C_VEL
LIN {X 0,Y 185.974,Z 321.943,A -85,B 0,C 180,E1 -22311.306,E2 -22311.306} C_VEL
LIN {X 0,Y 186.203,Z 321.915,A -85,B 0,C 180,E1 -22317.837,E2 -22317.837} C_VEL
LIN {X 0,Y 186.399,Z 321.891,A -85,B 0,C 180,E1 -22320,E2 -22320} C_VEL
LIN {X 0,Y 185.912,Z 321.953,A -85,B 0,C 180,E1 -22324.336,E2 -22324.336} C_VEL
LIN {X 0,Y 185.976,Z 321.944,A -85,B 0,C 180,E1 -22328.694,E2 -22328.694} C_VEL
LIN {X 0,Y 185.729,Z 321.977,A -85,B 0,C 180,E1 -22333.123,E2 -22333.123} C_VEL
LIN {X 0,Y 185.726,Z 322.088,A -85,B 0,C 180,E1 -22337.621,E2 -22337.621} C_VEL
LIN {X 0,Y 185.767,Z 323.093,A -85,B 0,C 180,E1 -22340.991,E2 -22340.991} C_VEL
LIN {X 0,Y 186.799,Z 325.788,A -85,B 0,C 180,E1 -22342.1,E2 -22342.1} C_VEL
LIN {X 0,Y 189.399,Z 328.786,A -85,B 0,C 180,E1 -22344.281,E2 -22344.281} C_VEL
LIN {X 0,Y 190.652,Z 329.939,A -85,B 0,C 180,E1 -22345.219,E2 -22345.219} C_VEL
LIN {X 0,Y 192.538,Z 333.527,A -85,B 0,C 180,E1 -22346.78,E2 -22346.78} C_VEL
LIN {X 0,Y 194.838,Z 336.191,A -85,B 0,C 180,E1 -22348.404,E2 -22348.404} C_VEL
LIN {X 0,Y 196.977,Z 340.008,A -85,B 0,C 180,E1 -22349.967,E2 -22349.967} C_VEL
LIN {X 0,Y 198.449,Z 342.086,A -85,B 0,C 180,E1 -22350.972,E2 -22350.972} C_VEL
LIN {X 0,Y 200.951,Z 346.345,A -85,B 0,C 180,E1 -22352.678,E2 -22352.678} C_VEL
LIN {X 0,Y 204.425,Z 353.083,A -85,B 0,C 180,E1 -22355.084,E2 -22355.084} C_VEL
LIN {X 0,Y 209.214,Z 363.418,A -85,B 0,C 180,E1 -22358.423,E2 -22358.423} C_VEL
LIN {X 0,Y 212.263,Z 373.023,A -85,B 0,C 180,E1 -22361.056,E2 -22361.056} C_VEL
LIN {X 0,Y 213.962,Z 381.761,A -85,B 0,C 180,E1 -22363.191,E2 -22363.191} C_VEL
LIN {X 0,Y 215.174,Z 392.442,A -85,B 0,C 180,E1 -22365.722,E2 -22365.722} C_VEL
LIN {X 0,Y 215.391,Z 404.627,A -85,B 0,C 180,E1 -22368.631,E2 -22368.631} C_VEL
LIN {X 0,Y 215.179,Z 408.247,A -85,B 0,C 180,E1 -22369.523,E2 -22369.523} C_VEL
LIN {X 0,Y 210.275,Z 420.046,A -85,B 0,C 180,E1 -22371.806,E2 -22371.806} C_VEL
LIN {X 0,Y 205.354,Z 430.857,A -85,B 0,C 180,E1 -22374.422,E2 -22374.422} C_VEL
LIN {X 0,Y 200.508,Z 440.774,A -85,B 0,C 180,E1 -22377.42,E2 -22377.42} C_VEL
LIN {X 0,Y 196.462,Z 449.027,A -85,B 0,C 180,E1 -22380.536,E2 -22380.536} C_VEL
LIN {X 0,Y 192.485,Z 456.491,A -85,B 0,C 180,E1 -22384.014,E2 -22384.014} C_VEL
LIN {X 0,Y 188.828,Z 463.451,A -85,B 0,C 180,E1 -22388.149,E2 -22388.149} C_VEL
LIN {X 0,Y 186.22,Z 468.925,A -85,B 0,C 180,E1 -22392.426,E2 -22392.426} C_VEL
LIN {X 0,Y 185.913,Z 469.599,A -85,B 0,C 180,E1 -22393.056,E2 -22393.056} C_VEL
LIN {X 0,Y 184.501,Z 471.362,A -85,B 0,C 180,E1 -22394.746,E2 -22394.746} C_VEL
LIN {X 0,Y 180.636,Z 473.811,A -85,B 0,C 180,E1 -22397.51,E2 -22397.51} C_VEL
LIN {X 0,Y 177.621,Z 475.375,A -85,B 0,C 180,E1 -22399.821,E2 -22399.821} C_VEL
LIN {X 0,Y 176.271,Z 476.309,A -85,B 0,C 180,E1 -22401.668,E2 -22401.668} C_VEL
LIN {X 0,Y 176.114,Z 476.544,A -85,B 0,C 180,E1 -22402.302,E2 -22402.302} C_VEL
LIN {X 0,Y 175.934,Z 477.625,A -85,B 0,C 180,E1 -22405.417,E2 -22405.417} C_VEL
LIN {X 0,Y 175.971,Z 478.216,A -85,B 0,C 180,E1 -22409.999,E2 -22409.999} C_VEL
LIN {X 0,Y 175.933,Z 477.609,A -85,B 0,C 180,E1 -22414.582,E2 -22414.582} C_VEL
LIN {X 0,Y 176.327,Z 475.86,A -85,B 0,C 180,E1 -22419.173,E2 -22419.173} C_VEL
LIN {X 0,Y 177.382,Z 472.943,A -85,B 0,C 180,E1 -22423.751,E2 -22423.751} C_VEL
LIN {X 0,Y 179.392,Z 468.793,A -85,B 0,C 180,E1 -22428.264,E2 -22428.264} C_VEL
LIN {X 0,Y 182.22,Z 463.296,A -85,B 0,C 180,E1 -22432.685,E2 -22432.685} C_VEL
LIN {X 0,Y 186.042,Z 456.304,A -85,B 0,C 180,E1 -22436.955,E2 -22436.955} C_VEL
LIN {X 0,Y 190.277,Z 448.828,A -85,B 0,C 180,E1 -22440.52,E2 -22440.52} C_VEL
LIN {X 0,Y 195.126,Z 439.525,A -85,B 0,C 180,E1 -22444.065,E2 -22444.065} C_VEL
LIN {X 0,Y 200.416,Z 428.971,A -85,B 0,C 180,E1 -22447.22,E2 -22447.22} C_VEL
LIN {X 0,Y 205.616,Z 417.808,A -85,B 0,C 180,E1 -22449.856,E2 -22449.856} C_VEL
LIN {X 0,Y 209.094,Z 409.528,A -85,B 0,C 180,E1 -22451.473,E2 -22451.473} C_VEL
LIN {X 0,Y 209.427,Z 399.79,A -85,B 0,C 180,E1 -22453.959,E2 -22453.959} C_VEL
LIN {X 0,Y 209.011,Z 390.124,A -85,B 0,C 180,E1 -22456.372,E2 -22456.372} C_VEL
LIN {X 0,Y 208.036,Z 381.901,A -85,B 0,C 180,E1 -22458.439,E2 -22458.439} C_VEL
LIN {X 0,Y 206.6,Z 374.567,A -85,B 0,C 180,E1 -22460.37,E2 -22460.37} C_VEL
LIN {X 0,Y 204.528,Z 367.835,A -85,B 0,C 180,E1 -22462.353,E2 -22462.353} C_VEL
LIN {X 0,Y 201.425,Z 360.356,A -85,B 0,C 180,E1 -22464.851,E2 -22464.851} C_VEL
LIN {X 0,Y 197.204,Z 351.662,A -85,B 0,C 180,E1 -22468.1,E2 -22468.1} C_VEL
LIN {X 0,Y 194.489,Z 346.672,A -85,B 0,C 180,E1 -22470.214,E2 -22470.214} C_VEL
LIN {X 0,Y 192.275,Z 343.025,A -85,B 0,C 180,E1 -22471.927,E2 -22471.927} C_VEL
LIN {X 0,Y 191.506,Z 341.559,A -85,B 0,C 180,E1 -22472.584,E2 -22472.584} C_VEL
LIN {X 0,Y 189.2,Z 338.423,A -85,B 0,C 180,E1 -22474.434,E2 -22474.434} C_VEL
LIN {X 0,Y 187.987,Z 335.871,A -85,B 0,C 180,E1 -22475.57,E2 -22475.57} C_VEL
LIN {X 0,Y 185.084,Z 332.649,A -85,B 0,C 180,E1 -22478.124,E2 -22478.124} C_VEL
LIN {X 0,Y 183.64,Z 329.544,A -85,B 0,C 180,E1 -22479.707,E2 -22479.707} C_VEL
LIN {X 0,Y 180.045,Z 326.348,A -85,B 0,C 180,E1 -22483.561,E2 -22483.561} C_VEL
LIN {X 0,Y 178.807,Z 323.764,A -85,B 0,C 180,E1 -22485.416,E2 -22485.416} C_VEL
LIN {X 0,Y 178.637,Z 322.855,A -85,B 0,C 180,E1 -22485.911,E2 -22485.911} C_VEL
LIN {X 0,Y 178.899,Z 322.82,A -85,B 0,C 180,E1 -22490.959,E2 -22490.959} C_VEL
LIN {X 0,Y 179.144,Z 322.788,A -85,B 0,C 180,E1 -22497.752,E2 -22497.752} C_VEL
LIN {X 0,Y 179.36,Z 322.768,A -85,B 0,C 180,E1 -22500,E2 -22500} C_VEL
LIN {X 0,Y 178.854,Z 322.831,A -85,B 0,C 180,E1 -22504.508,E2 -22504.508} C_VEL
LIN {X 0,Y 178.899,Z 322.82,A -85,B 0,C 180,E1 -22509.041,E2 -22509.041} C_VEL
LIN {X 0,Y 178.648,Z 323.017,A -85,B 0,C 180,E1 -22514.452,E2 -22514.452} C_VEL
LIN {X 0,Y 179.504,Z 325.476,A -85,B 0,C 180,E1 -22515.907,E2 -22515.907} C_VEL
LIN {X 0,Y 181.759,Z 327.883,A -85,B 0,C 180,E1 -22518.601,E2 -22518.601} C_VEL
LIN {X 0,Y 183.647,Z 329.03,A -85,B 0,C 180,E1 -22520.439,E2 -22520.439} C_VEL
LIN {X 0,Y 184.954,Z 331.759,A -85,B 0,C 180,E1 -22521.892,E2 -22521.892} C_VEL
LIN {X 0,Y 187.96,Z 334.709,A -85,B 0,C 180,E1 -22524.506,E2 -22524.506} C_VEL
LIN {X 0,Y 190.186,Z 338.561,A -85,B 0,C 180,E1 -22526.472,E2 -22526.472} C_VEL
LIN {X 0,Y 191.837,Z 340.625,A -85,B 0,C 180,E1 -22527.772,E2 -22527.772} C_VEL
LIN {X 0,Y 194.215,Z 344.666,A -85,B 0,C 180,E1 -22529.671,E2 -22529.671} C_VEL
LIN {X 0,Y 195.21,Z 346.207,A -85,B 0,C 180,E1 -22530.417,E2 -22530.417} C_VEL
LIN {X 0,Y 198.131,Z 351.659,A -85,B 0,C 180,E1 -22532.691,E2 -22532.691} C_VEL
LIN {X 0,Y 201.989,Z 359.462,A -85,B 0,C 180,E1 -22535.648,E2 -22535.648} C_VEL
LIN {X 0,Y 205.579,Z 368.329,A -85,B 0,C 180,E1 -22538.602,E2 -22538.602} C_VEL
LIN {X 0,Y 207.669,Z 375.604,A -85,B 0,C 180,E1 -22540.732,E2 -22540.732} C_VEL
LIN {X 0,Y 209.278,Z 384.733,A -85,B 0,C 180,E1 -22543.176,E2 -22543.176} C_VEL
LIN {X 0,Y 210.224,Z 395.513,A -85,B 0,C 180,E1 -22545.952,E2 -22545.952} C_VEL
LIN {X 0,Y 210.241,Z 404.708,A -85,B 0,C 180,E1 -22548.366,E2 -22548.366} C_VEL
LIN {X 0,Y 205.271,Z 416.541,A -85,B 0,C 180,E1 -22550.7,E2 -22550.7} C_VEL
LIN {X 0,Y 200.201,Z 427.373,A -85,B 0,C 180,E1 -22553.362,E2 -22553.362} C_VEL
LIN {X 0,Y 194.974,Z 437.909,A -85,B 0,C 180,E1 -22556.655,E2 -22556.655} C_VEL
LIN {X 0,Y 190.142,Z 446.67,A -85,B 0,C 180,E1 -22560.069,E2 -22560.069} C_VEL
LIN {X 0,Y 186.649,Z 452.998,A -85,B 0,C 180,E1 -22563.139,E2 -22563.139} C_VEL
LIN {X 0,Y 182.764,Z 459.96,A -85,B 0,C 180,E1 -22567.386,E2 -22567.386} C_VEL
LIN {X 0,Y 179.849,Z 465.428,A -85,B 0,C 180,E1 -22571.784,E2 -22571.784} C_VEL
LIN {X 0,Y 177.742,Z 469.555,A -85,B 0,C 180,E1 -22576.277,E2 -22576.277} C_VEL
LIN {X 0,Y 176.537,Z 472.451,A -85,B 0,C 180,E1 -22580.838,E2 -22580.838} C_VEL
LIN {X 0,Y 176.009,Z 474.189,A -85,B 0,C 180,E1 -22585.42,E2 -22585.42} C_VEL
LIN {X 0,Y 175.981,Z 474.793,A -85,B 0,C 180,E1 -22590.001,E2 -22590.001} C_VEL
LIN {X 0,Y 176.009,Z 474.223,A -85,B 0,C 180,E1 -22594.581,E2 -22594.581} C_VEL
LIN {X 0,Y 176.528,Z 472.53,A -85,B 0,C 180,E1 -22599.164,E2 -22599.164} C_VEL
LIN {X 0,Y 177.719,Z 469.674,A -85,B 0,C 180,E1 -22603.726,E2 -22603.726} C_VEL
LIN {X 0,Y 179.806,Z 465.587,A -85,B 0,C 180,E1 -22608.222,E2 -22608.222} C_VEL
LIN {X 0,Y 182.672,Z 460.17,A -85,B 0,C 180,E1 -22612.628,E2 -22612.628} C_VEL
LIN {X 0,Y 186.575,Z 453.266,A -85,B 0,C 180,E1 -22616.874,E2 -22616.874} C_VEL
LIN {X 0,Y 191.36,Z 444.652,A -85,B 0,C 180,E1 -22620.943,E2 -22620.943} C_VEL
LIN {X 0,Y 195.907,Z 436.185,A -85,B 0,C 180,E1 -22624.111,E2 -22624.111} C_VEL
LIN {X 0,Y 200.937,Z 426.167,A -85,B 0,C 180,E1 -22627.11,E2 -22627.11} C_VEL
LIN {X 0,Y 206.464,Z 414.094,A -85,B 0,C 180,E1 -22629.979,E2 -22629.979} C_VEL
LIN {X 0,Y 210.17,Z 405.297,A -85,B 0,C 180,E1 -22631.653,E2 -22631.653} C_VEL
LIN {X 0,Y 210.336,Z 395.693,A -85,B 0,C 180,E1 -22634.143,E2 -22634.143} C_VEL
LIN {X 0,Y 209.431,Z 385.157,A -85,B 0,C 180,E1 -22636.863,E2 -22636.863} C_VEL
LIN {X 0,Y 207.68,Z 375.32,A -85,B 0,C 180,E1 -22639.512,E2 -22639.512} C_VEL
LIN {X 0,Y 205.144,Z 367.006,A -85,B 0,C 180,E1 -22641.995,E2 -22641.995} C_VEL
LIN {X 0,Y 201.576,Z 358.516,A -85,B 0,C 180,E1 -22644.881,E2 -22644.881} C_VEL
LIN {X 0,Y 199.01,Z 353.329,A -85,B 0,C 180,E1 -22646.867,E2 -22646.867} C_VEL
LIN {X 0,Y 197.081,Z 349.611,A -85,B 0,C 180,E1 -22648.34,E2 -22648.34} C_VEL
LIN {X 0,Y 194.518,Z 345.016,A -85,B 0,C 180,E1 -22650.361,E2 -22650.361} C_VEL
LIN {X 0,Y 192.071,Z 341.167,A -85,B 0,C 180,E1 -22652.264,E2 -22652.264} C_VEL
LIN {X 0,Y 191.256,Z 339.798,A -85,B 0,C 180,E1 -22652.952,E2 -22652.952} C_VEL
LIN {X 0,Y 188.604,Z 336.181,A -85,B 0,C 180,E1 -22655.141,E2 -22655.141} C_VEL
LIN {X 0,Y 187.644,Z 334.319,A -85,B 0,C 180,E1 -22656.054,E2 -22656.054} C_VEL
LIN {X 0,Y 184.91,Z 331.724,A -85,B 0,C 180,E1 -22658.468,E2 -22658.468} C_VEL
LIN {X 0,Y 183.462,Z 328.747,A -85,B 0,C 180,E1 -22660.099,E2 -22660.099} C_VEL
LIN {X 0,Y 180.413,Z 326.765,A -85,B 0,C 180,E1 -22663.304,E2 -22663.304} C_VEL
LIN {X 0,Y 178.905,Z 324.093,A -85,B 0,C 180,E1 -22665.497,E2 -22665.497} C_VEL
LIN {X 0,Y 178.649,Z 322.852,A -85,B 0,C 180,E1 -22666.129,E2 -22666.129} C_VEL
LIN {X 0,Y 178.905,Z 322.825,A -85,B 0,C 180,E1 -22670.959,E2 -22670.959} C_VEL
LIN {X 0,Y 179.149,Z 322.793,A -85,B 0,C 180,E1 -22677.751,E2 -22677.751} C_VEL
LIN {X 0,Y 179.363,Z 322.768,A -85,B 0,C 180,E1 -22680,E2 -22680} C_VEL
LIN {X 0,Y 178.859,Z 322.831,A -85,B 0,C 180,E1 -22684.507,E2 -22684.507} C_VEL
LIN {X 0,Y 178.906,Z 322.824,A -85,B 0,C 180,E1 -22689.04,E2 -22689.04} C_VEL
LIN {X 0,Y 178.653,Z 322.893,A -85,B 0,C 180,E1 -22693.87,E2 -22693.87} C_VEL
LIN {X 0,Y 179.305,Z 325.073,A -85,B 0,C 180,E1 -22695.05,E2 -22695.05} C_VEL
LIN {X 0,Y 181.182,Z 327.544,A -85,B 0,C 180,E1 -22697.495,E2 -22697.495} C_VEL
LIN {X 0,Y 183.847,Z 329.936,A -85,B 0,C 180,E1 -22700.269,E2 -22700.269} C_VEL
LIN {X 0,Y 185.283,Z 332.954,A -85,B 0,C 180,E1 -22701.851,E2 -22701.851} C_VEL
LIN {X 0,Y 188.239,Z 336.335,A -85,B 0,C 180,E1 -22704.468,E2 -22704.468} C_VEL
LIN {X 0,Y 190.451,Z 340.327,A -85,B 0,C 180,E1 -22706.431,E2 -22706.431} C_VEL
LIN {X 0,Y 191.959,Z 342.173,A -85,B 0,C 180,E1 -22707.604,E2 -22707.604} C_VEL
LIN {X 0,Y 194.154,Z 346.23,A -85,B 0,C 180,E1 -22709.402,E2 -22709.402} C_VEL
LIN {X 0,Y 195.33,Z 348.108,A -85,B 0,C 180,E1 -22710.286,E2 -22710.286} C_VEL
LIN {X 0,Y 198.24,Z 353.678,A -85,B 0,C 180,E1 -22712.558,E2 -22712.558} C_VEL
LIN {X 0,Y 201.557,Z 360.569,A -85,B 0,C 180,E1 -22715.123,E2 -22715.123} C_VEL
LIN {X 0,Y 205.177,Z 369.48,A -85,B 0,C 180,E1 -22718.065,E2 -22718.065} C_VEL
LIN {X 0,Y 207.471,Z 378.125,A -85,B 0,C 180,E1 -22720.504,E2 -22720.504} C_VEL
LIN {X 0,Y 208.805,Z 386.983,A -85,B 0,C 180,E1 -22722.786,E2 -22722.786} C_VEL
LIN {X 0,Y 209.53,Z 396.663,A -85,B 0,C 180,E1 -22725.221,E2 -22725.221} C_VEL
LIN {X 0,Y 209.385,Z 406.996,A -85,B 0,C 180,E1 -22727.832,E2 -22727.832} C_VEL
LIN {X 0,Y 209.211,Z 409.619,A -85,B 0,C 180,E1 -22728.507,E2 -22728.507} C_VEL
LIN {X 0,Y 204.726,Z 419.98,A -85,B 0,C 180,E1 -22730.574,E2 -22730.574} C_VEL
LIN {X 0,Y 199.595,Z 430.79,A -85,B 0,C 180,E1 -22733.231,E2 -22733.231} C_VEL
LIN {X 0,Y 194.195,Z 441.302,A -85,B 0,C 180,E1 -22736.495,E2 -22736.495} C_VEL
LIN {X 0,Y 190.268,Z 448.959,A -85,B 0,C 180,E1 -22739.476,E2 -22739.476} C_VEL
LIN {X 0,Y 186.052,Z 456.422,A -85,B 0,C 180,E1 -22743.044,E2 -22743.044} C_VEL
LIN {X 0,Y 182.196,Z 463.383,A -85,B 0,C 180,E1 -22747.31,E2 -22747.31} C_VEL
LIN {X 0,Y 179.388,Z 468.856,A -85,B 0,C 180,E1 -22751.734,E2 -22751.734} C_VEL
LIN {X 0,Y 177.383,Z 472.994,A -85,B 0,C 180,E1 -22756.247,E2 -22756.247} C_VEL
LIN {X 0,Y 176.328,Z 475.895,A -85,B 0,C 180,E1 -22760.825,E2 -22760.825} C_VEL
LIN {X 0,Y 176.114,Z 476.544,A -85,B 0,C 180,E1 -22762.302,E2 -22762.302} C_VEL
LIN {X 0,Y 175.31,Z 477.287,A -85,B 0,C 180,E1 -22764.194,E2 -22764.194} C_VEL
LIN {X 0,Y 173.681,Z 477.826,A -85,B 0,C 180,E1 -22766.063,E2 -22766.063} C_VEL
LIN {X 0,Y 169.975,Z 478.232,A -85,B 0,C 180,E1 -22769.869,E2 -22769.869} C_VEL
LIN {X 0,Y 168.914,Z 478.072,A -85,B 0,C 180,E1 -22771.863,E2 -22771.863} C_VEL
LIN {X 0,Y 168.811,Z 477.96,A -85,B 0,C 180,E1 -22772.539,E2 -22772.539} C_VEL
LIN {X 0,Y 168.964,Z 476.808,A -85,B 0,C 180,E1 -22777.167,E2 -22777.167} C_VEL
LIN {X 0,Y 169.764,Z 474.481,A -85,B 0,C 180,E1 -22781.945,E2 -22781.945} C_VEL
LIN {X 0,Y 171.447,Z 470.958,A -85,B 0,C 180,E1 -22786.674,E2 -22786.674} C_VEL
LIN {X 0,Y 173.991,Z 466.15,A -85,B 0,C 180,E1 -22791.316,E2 -22791.316} C_VEL
LIN {X 0,Y 177.53,Z 459.927,A -85,B 0,C 180,E1 -22795.813,E2 -22795.813} C_VEL
LIN {X 0,Y 182.076,Z 452.114,A -85,B 0,C 180,E1 -22800.117,E2 -22800.117} C_VEL
LIN {X 0,Y 186.912,Z 443.807,A -85,B 0,C 180,E1 -22803.682,E2 -22803.682} C_VEL
LIN {X 0,Y 192.249,Z 433.794,A -85,B 0,C 180,E1 -22807.097,E2 -22807.097} C_VEL
LIN {X 0,Y 197.388,Z 423.559,A -85,B 0,C 180,E1 -22809.856,E2 -22809.856} C_VEL
LIN {X 0,Y 203.1,Z 411.179,A -85,B 0,C 180,E1 -22812.487,E2 -22812.487} C_VEL
LIN {X 0,Y 203.66,Z 401.166,A -85,B 0,C 180,E1 -22815.15,E2 -22815.15} C_VEL
LIN {X 0,Y 203.393,Z 391.695,A -85,B 0,C 180,E1 -22817.668,E2 -22817.668} C_VEL
LIN {X 0,Y 202.426,Z 382.854,A -85,B 0,C 180,E1 -22820.035,E2 -22820.035} C_VEL
LIN {X 0,Y 200.726,Z 374.932,A -85,B 0,C 180,E1 -22822.345,E2 -22822.345} C_VEL
LIN {X 0,Y 197.619,Z 366.251,A -85,B 0,C 180,E1 -22825.319,E2 -22825.319} C_VEL
LIN {X 0,Y 193.602,Z 357.257,A -85,B 0,C 180,E1 -22828.849,E2 -22828.849} C_VEL
LIN {X 0,Y 191.122,Z 352.383,A -85,B 0,C 180,E1 -22831.01,E2 -22831.01} C_VEL
LIN {X 0,Y 188.981,Z 348.249,A -85,B 0,C 180,E1 -22832.974,E2 -22832.974} C_VEL
LIN {X 0,Y 186.273,Z 344.045,A -85,B 0,C 180,E1 -22835.405,E2 -22835.405} C_VEL
LIN {X 0,Y 185.207,Z 341.925,A -85,B 0,C 180,E1 -22836.52,E2 -22836.52} C_VEL
LIN {X 0,Y 182.592,Z 338.471,A -85,B 0,C 180,E1 -22839.143,E2 -22839.143} C_VEL
LIN {X 0,Y 181.385,Z 336.002,A -85,B 0,C 180,E1 -22840.606,E2 -22840.606} C_VEL
LIN {X 0,Y 177.981,Z 332.249,A -85,B 0,C 180,E1 -22844.835,E2 -22844.835} C_VEL
LIN {X 0,Y 177.053,Z 329.746,A -85,B 0,C 180,E1 -22846.514,E2 -22846.514} C_VEL
LIN {X 0,Y 172.842,Z 326.28,A -85,B 0,C 180,E1 -22857.087,E2 -22857.087} C_VEL
LIN {X 0,Y 172.742,Z 325.326,A -85,B 0,C 180,E1 -22860,E2 -22860} C_VEL
LIN {X 0,Y 177.126,Z 330.031,A -85,B 0,C 180,E1 -22873.846,E2 -22873.846} C_VEL
LIN {X 0,Y 178.362,Z 332.89,A -85,B 0,C 180,E1 -22876.011,E2 -22876.011} C_VEL
LIN {X 0,Y 180.831,Z 335.163,A -85,B 0,C 180,E1 -22878.995,E2 -22878.995} C_VEL
LIN {X 0,Y 181.594,Z 335.755,A -85,B 0,C 180,E1 -22879.794,E2 -22879.794} C_VEL
LIN {X 0,Y 183.192,Z 338.758,A -85,B 0,C 180,E1 -22881.67,E2 -22881.67} C_VEL
LIN {X 0,Y 185.516,Z 341.237,A -85,B 0,C 180,E1 -22883.884,E2 -22883.884} C_VEL
LIN {X 0,Y 187.934,Z 345.362,A -85,B 0,C 180,E1 -22886.204,E2 -22886.204} C_VEL
LIN {X 0,Y 188.949,Z 346.812,A -85,B 0,C 180,E1 -22887.097,E2 -22887.097} C_VEL
LIN {X 0,Y 191.304,Z 350.935,A -85,B 0,C 180,E1 -22889.197,E2 -22889.197} C_VEL
LIN {X 0,Y 195.887,Z 360.089,A -85,B 0,C 180,E1 -22893.171,E2 -22893.171} C_VEL
LIN {X 0,Y 199.767,Z 369.687,A -85,B 0,C 180,E1 -22896.733,E2 -22896.733} C_VEL
LIN {X 0,Y 201.772,Z 376.055,A -85,B 0,C 180,E1 -22898.827,E2 -22898.827} C_VEL
LIN {X 0,Y 203.294,Z 383.626,A -85,B 0,C 180,E1 -22901.06,E2 -22901.06} C_VEL
LIN {X 0,Y 204.292,Z 393.326,A -85,B 0,C 180,E1 -22903.746,E2 -22903.746} C_VEL
LIN {X 0,Y 204.445,Z 403.624,A -85,B 0,C 180,E1 -22906.568,E2 -22906.568} C_VEL
LIN {X 0,Y 204.349,Z 406.118,A -85,B 0,C 180,E1 -22907.264,E2 -22907.264} C_VEL
LIN {X 0,Y 199.796,Z 416.614,A -85,B 0,C 180,E1 -22909.403,E2 -22909.403} C_VEL
LIN {X 0,Y 194.524,Z 427.445,A -85,B 0,C 180,E1 -22912.108,E2 -22912.108} C_VEL
LIN {X 0,Y 189.752,Z 436.714,A -85,B 0,C 180,E1 -22915.006,E2 -22915.006} C_VEL
LIN {X 0,Y 184.653,Z 445.621,A -85,B 0,C 180,E1 -22918.446,E2 -22918.446} C_VEL
LIN {X 0,Y 180.301,Z 453.069,A -85,B 0,C 180,E1 -22922.113,E2 -22922.113} C_VEL
LIN {X 0,Y 176.023,Z 460.304,A -85,B 0,C 180,E1 -22926.681,E2 -22926.681} C_VEL
LIN {X 0,Y 173.083,Z 465.499,A -85,B 0,C 180,E1 -22931.046,E2 -22931.046} C_VEL
LIN {X 0,Y 170.817,Z 469.625,A -85,B 0,C 180,E1 -22935.709,E2 -22935.709} C_VEL
LIN {X 0,Y 169.504,Z 472.521,A -85,B 0,C 180,E1 -22940.455,E2 -22940.455} C_VEL
LIN {X 0,Y 168.932,Z 474.258,A -85,B 0,C 180,E1 -22945.228,E2 -22945.228} C_VEL
LIN {X 0,Y 168.88,Z 474.862,A -85,B 0,C 180,E1 -22950.001,E2 -22950.001} C_VEL
LIN {X 0,Y 168.932,Z 474.292,A -85,B 0,C 180,E1 -22954.774,E2 -22954.774} C_VEL
LIN {X 0,Y 169.496,Z 472.599,A -85,B 0,C 180,E1 -22959.548,E2 -22959.548} C_VEL
LIN {X 0,Y 170.775,Z 469.743,A -85,B 0,C 180,E1 -22964.296,E2 -22964.296} C_VEL
LIN {X 0,Y 173.036,Z 465.655,A -85,B 0,C 180,E1 -22968.962,E2 -22968.962} C_VEL
LIN {X 0,Y 176.112,Z 460.238,A -85,B 0,C 180,E1 -22973.52,E2 -22973.52} C_VEL
LIN {X 0,Y 180.214,Z 453.334,A -85,B 0,C 180,E1 -22977.904,E2 -22977.904} C_VEL
LIN {X 0,Y 185.297,Z 444.719,A -85,B 0,C 180,E1 -22982.073,E2 -22982.073} C_VEL
LIN {X 0,Y 190.301,Z 435.685,A -85,B 0,C 180,E1 -22985.513,E2 -22985.513} C_VEL
LIN {X 0,Y 195.302,Z 426.234,A -85,B 0,C 180,E1 -22988.371,E2 -22988.371} C_VEL
LIN {X 0,Y 201.052,Z 414.16,A -85,B 0,C 180,E1 -22991.285,E2 -22991.285} C_VEL
LIN {X 0,Y 204.352,Z 406.596,A -85,B 0,C 180,E1 -22992.766,E2 -22992.766} C_VEL
LIN {X 0,Y 204.563,Z 397.619,A -85,B 0,C 180,E1 -22995.228,E2 -22995.228} C_VEL
LIN {X 0,Y 203.769,Z 386.709,A -85,B 0,C 180,E1 -22998.241,E2 -22998.241} C_VEL
LIN {X 0,Y 202.381,Z 378.201,A -85,B 0,C 180,E1 -23000.671,E2 -23000.671} C_VEL
LIN {X 0,Y 200.693,Z 372.061,A -85,B 0,C 180,E1 -23002.615,E2 -23002.615} C_VEL
